Yaskawa INFORM job: A_ROOF_UPPER_0614_2_PAINT_25.JBI

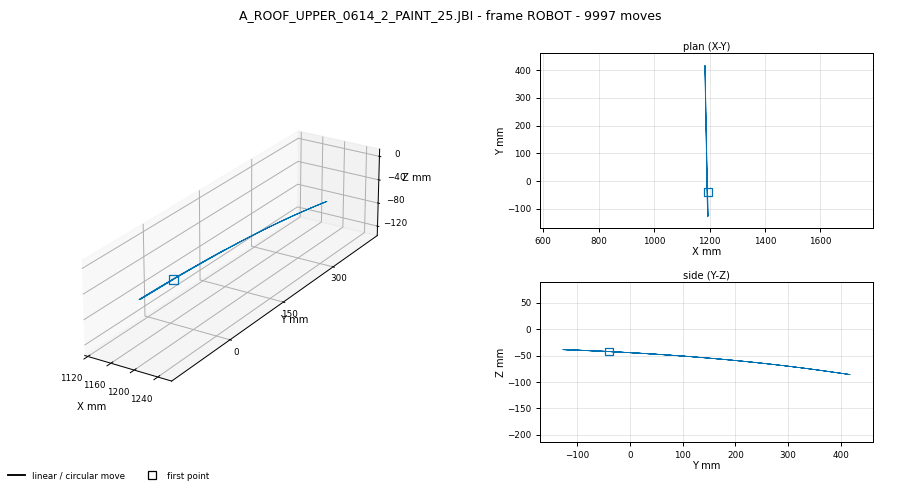
[picture p0: tool path of A_ROOF_UPPER_0614_2_PAINT_25.JBI in frame ROBOT, 9997 of 9997 moves have a stored position in this frame; points joined in program order, loops and branches not executed]
/JOB
//NAME A_ROOF_UPPER_0614_2_PAINT25
//POS
///NPOS 9997,0,0,0,0,0
///TOOL 1
///USER 0
///POSTYPE ROBOT
///RECTAN
///RCONF 1,0,0,0,0,0,0,0,0,0,0,0,0,0,0,0,0,0,0,0,0,0,0,0
C00000=1193.053,-39.607,-42.064,179.756,5.637,149.068
C00001=1193.058,-39.856,-42.051,179.753,5.636,149.068
C00002=1193.063,-40.106,-42.040,179.751,5.637,149.069
C00003=1193.068,-40.356,-42.027,179.748,5.636,149.070
C00004=1193.073,-40.606,-42.015,179.746,5.635,149.070
C00005=1193.078,-40.855,-42.002,179.744,5.636,149.071
C00006=1193.083,-41.105,-41.991,179.741,5.635,149.072
C00007=1193.088,-41.354,-41.978,179.739,5.635,149.072
C00008=1193.094,-41.604,-41.966,179.737,5.634,149.073
C00009=1193.099,-41.854,-41.954,179.735,5.634,149.074
C00010=1193.104,-42.104,-41.942,179.732,5.634,149.074
C00011=1193.110,-42.354,-41.930,179.729,5.634,149.075
C00012=1193.114,-42.603,-41.918,179.727,5.633,149.076
C00013=1193.119,-42.852,-41.906,179.725,5.633,149.076
C00014=1193.124,-43.102,-41.893,179.722,5.633,149.077
C00015=1193.130,-43.352,-41.882,179.720,5.632,149.078
C00016=1193.135,-43.602,-41.870,179.717,5.632,149.078
C00017=1193.140,-43.851,-41.857,179.715,5.632,149.079
C00018=1193.145,-44.101,-41.846,179.713,5.631,149.079
C00019=1193.151,-44.351,-41.834,179.710,5.631,149.080
C00020=1193.156,-44.600,-41.821,179.708,5.631,149.081
C00021=1193.161,-44.850,-41.809,179.705,5.631,149.082
C00022=1193.166,-45.099,-41.798,179.703,5.630,149.082
C00023=1193.171,-45.349,-41.786,179.700,5.629,149.083
C00024=1193.176,-45.599,-41.774,179.698,5.630,149.083
C00025=1193.182,-45.849,-41.762,179.696,5.629,149.084
C00026=1193.187,-46.098,-41.749,179.694,5.629,149.085
C00027=1193.192,-46.348,-41.738,179.691,5.629,149.085
C00028=1193.197,-46.597,-41.726,179.689,5.628,149.086
C00029=1193.202,-46.847,-41.713,179.686,5.628,149.087
C00030=1193.208,-47.097,-41.702,179.683,5.628,149.087
C00031=1193.212,-47.346,-41.690,179.682,5.628,149.088
C00032=1193.218,-47.596,-41.678,179.679,5.627,149.089
C00033=1193.223,-47.846,-41.666,179.677,5.627,149.089
C00034=1193.228,-48.095,-41.654,179.674,5.627,149.090
C00035=1193.233,-48.345,-41.643,179.672,5.626,149.091
C00036=1193.239,-48.594,-41.631,179.670,5.626,149.091
C00037=1193.244,-48.844,-41.619,179.667,5.625,149.092
C00038=1193.250,-49.115,-41.606,179.665,5.626,149.093
C00039=1193.255,-49.385,-41.593,179.662,5.625,149.093
C00040=1193.261,-49.655,-41.581,179.660,5.625,149.094
C00041=1193.266,-49.925,-41.568,179.657,5.624,149.095
C00042=1193.271,-50.175,-41.556,179.654,5.624,149.095
C00043=1193.276,-50.425,-41.545,179.652,5.624,149.096
C00044=1193.282,-50.674,-41.532,179.650,5.623,149.097
C00045=1193.286,-50.924,-41.521,179.647,5.623,149.097
C00046=1193.292,-51.174,-41.509,179.645,5.623,149.098
C00047=1193.298,-51.423,-41.497,179.643,5.623,149.099
C00048=1193.302,-51.672,-41.486,179.640,5.622,149.099
C00049=1193.308,-51.922,-41.474,179.638,5.622,149.100
C00050=1193.313,-52.172,-41.462,179.636,5.622,149.101
C00051=1193.318,-52.421,-41.450,179.633,5.622,149.101
C00052=1193.323,-52.671,-41.438,179.631,5.621,149.102
C00053=1193.328,-52.921,-41.426,179.629,5.621,149.102
C00054=1193.333,-53.171,-41.415,179.626,5.621,149.103
C00055=1193.339,-53.421,-41.403,179.623,5.620,149.104
C00056=1193.344,-53.670,-41.392,179.621,5.621,149.105
C00057=1193.349,-53.920,-41.380,179.619,5.620,149.105
C00058=1193.354,-54.169,-41.369,179.616,5.619,149.106
C00059=1193.359,-54.419,-41.357,179.614,5.620,149.106
C00060=1193.365,-54.669,-41.345,179.612,5.619,149.107
C00061=1193.370,-54.919,-41.334,179.609,5.618,149.108
C00062=1193.375,-55.169,-41.322,179.607,5.619,149.108
C00063=1193.380,-55.418,-41.311,179.605,5.618,149.109
C00064=1193.386,-55.667,-41.299,179.602,5.618,149.110
C00065=1193.390,-55.917,-41.288,179.600,5.617,149.110
C00066=1193.396,-56.167,-41.276,179.598,5.617,149.111
C00067=1193.401,-56.417,-41.265,179.595,5.617,149.112
C00068=1193.406,-56.667,-41.253,179.592,5.617,149.112
C00069=1193.411,-56.916,-41.242,179.590,5.617,149.113
C00070=1193.417,-57.165,-41.230,179.588,5.616,149.114
C00071=1193.422,-57.415,-41.218,179.586,5.616,149.114
C00072=1193.427,-57.665,-41.207,179.583,5.616,149.115
C00073=1193.432,-57.915,-41.195,179.581,5.616,149.116
C00074=1193.437,-58.165,-41.184,179.579,5.615,149.116
C00075=1193.443,-58.414,-41.172,179.577,5.615,149.117
C00076=1193.448,-58.663,-41.161,179.574,5.615,149.118
C00077=1193.452,-58.913,-41.150,179.571,5.614,149.118
C00078=1193.458,-59.163,-41.138,179.570,5.614,149.119
C00079=1193.462,-59.413,-41.127,179.567,5.614,149.119
C00080=1193.468,-59.662,-41.115,179.564,5.613,149.120
C00081=1193.473,-59.911,-41.104,179.562,5.614,149.121
C00082=1193.479,-60.162,-41.093,179.560,5.613,149.121
C00083=1193.484,-60.412,-41.081,179.557,5.613,149.122
C00084=1193.489,-60.662,-41.069,179.555,5.613,149.123
C00085=1193.494,-60.911,-41.058,179.553,5.612,149.123
C00086=1193.500,-61.160,-41.047,179.550,5.612,149.124
C00087=1193.504,-61.410,-41.035,179.548,5.612,149.125
C00088=1193.509,-61.660,-41.024,179.546,5.612,149.125
C00089=1193.515,-61.910,-41.013,179.543,5.611,149.126
C00090=1193.520,-62.159,-41.002,179.541,5.611,149.126
C00091=1193.526,-62.409,-40.990,179.539,5.611,149.127
C00092=1193.530,-62.659,-40.979,179.536,5.610,149.128
C00093=1193.536,-62.908,-40.967,179.534,5.611,149.129
C00094=1193.541,-63.158,-40.956,179.532,5.610,149.129
C00095=1193.546,-63.408,-40.945,179.530,5.610,149.130
C00096=1193.551,-63.658,-40.933,179.527,5.610,149.131
C00097=1193.557,-63.907,-40.923,179.524,5.609,149.131
C00098=1193.561,-64.156,-40.911,179.523,5.609,149.132
C00099=1193.567,-64.407,-40.900,179.520,5.609,149.132
C00100=1193.572,-64.656,-40.889,179.517,5.608,149.133
C00101=1193.578,-64.906,-40.877,179.515,5.609,149.134
C00102=1193.583,-65.155,-40.866,179.513,5.608,149.134
C00103=1193.588,-65.406,-40.855,179.511,5.608,149.135
C00104=1193.594,-65.655,-40.844,179.508,5.608,149.136
C00105=1193.598,-65.904,-40.833,179.506,5.607,149.136
C00106=1193.603,-66.154,-40.821,179.504,5.607,149.137
C00107=1193.609,-66.404,-40.811,179.502,5.607,149.138
C00108=1193.614,-66.654,-40.799,179.499,5.607,149.138
C00109=1193.619,-66.903,-40.788,179.496,5.606,149.139
C00110=1193.625,-67.153,-40.777,179.495,5.606,149.139
C00111=1193.630,-67.403,-40.766,179.492,5.606,149.140
C00112=1193.634,-67.652,-40.755,179.490,5.606,149.141
C00113=1193.641,-67.902,-40.744,179.487,5.606,149.142
C00114=1193.645,-68.152,-40.732,179.485,5.605,149.142
C00115=1193.650,-68.401,-40.721,179.483,5.605,149.143
C00116=1193.656,-68.651,-40.711,179.480,5.605,149.143
C00117=1193.661,-68.901,-40.699,179.478,5.604,149.144
C00118=1193.666,-69.151,-40.688,179.476,5.604,149.145
C00119=1193.671,-69.400,-40.678,179.473,5.604,149.145
C00120=1193.677,-69.650,-40.666,179.471,5.604,149.146
C00121=1193.682,-69.900,-40.655,179.469,5.604,149.147
C00122=1193.687,-70.149,-40.644,179.466,5.603,149.147
C00123=1193.692,-70.399,-40.633,179.464,5.603,149.148
C00124=1193.698,-70.649,-40.622,179.462,5.603,149.149
C00125=1193.703,-70.898,-40.611,179.459,5.603,149.149
C00126=1193.708,-71.149,-40.600,179.457,5.603,149.150
C00127=1193.713,-71.397,-40.589,179.455,5.602,149.151
C00128=1193.719,-71.648,-40.578,179.452,5.602,149.151
C00129=1193.724,-71.898,-40.567,179.450,5.602,149.152
C00130=1193.729,-72.147,-40.556,179.448,5.601,149.152
C00131=1193.734,-72.397,-40.545,179.446,5.602,149.153
C00132=1193.739,-72.646,-40.534,179.443,5.601,149.154
C00133=1193.745,-72.896,-40.523,179.441,5.600,149.154
C00134=1193.750,-73.146,-40.512,179.439,5.601,149.155
C00135=1193.755,-73.395,-40.502,179.436,5.600,149.156
C00136=1193.760,-73.645,-40.490,179.434,5.601,149.156
C00137=1193.765,-73.895,-40.480,179.432,5.600,149.157
C00138=1193.771,-74.145,-40.468,179.429,5.600,149.158
C00139=1193.776,-74.395,-40.458,179.427,5.600,149.158
C00140=1193.781,-74.644,-40.447,179.424,5.599,149.159
C00141=1193.786,-74.894,-40.436,179.422,5.599,149.160
C00142=1193.792,-75.164,-40.424,179.420,5.599,149.160
C00143=1193.798,-75.435,-40.412,179.417,5.599,149.161
C00144=1193.803,-75.707,-40.401,179.415,5.598,149.162
C00145=1193.809,-75.977,-40.389,179.412,5.598,149.162
C00146=1193.814,-76.227,-40.379,179.410,5.598,149.163
C00147=1193.820,-76.476,-40.368,179.407,5.598,149.164
C00148=1193.825,-76.726,-40.357,179.406,5.598,149.164
C00149=1193.830,-76.976,-40.345,179.403,5.597,149.165
C00150=1193.836,-77.226,-40.335,179.400,5.597,149.166
C00151=1193.841,-77.476,-40.325,179.399,5.597,149.166
C00152=1193.846,-77.725,-40.314,179.396,5.596,149.167
C00153=1193.851,-77.975,-40.303,179.394,5.597,149.168
C00154=1193.856,-78.224,-40.292,179.391,5.596,149.168
C00155=1193.861,-78.474,-40.282,179.389,5.596,149.169
C00156=1193.867,-78.724,-40.271,179.387,5.596,149.170
C00157=1193.872,-78.973,-40.260,179.384,5.596,149.170
C00158=1193.877,-79.223,-40.250,179.382,5.596,149.171
C00159=1193.882,-79.473,-40.239,179.380,5.595,149.171
C00160=1193.888,-79.722,-40.228,179.377,5.595,149.172
C00161=1193.893,-79.973,-40.217,179.375,5.595,149.173
C00162=1193.899,-80.222,-40.207,179.373,5.594,149.173
C00163=1193.904,-80.472,-40.196,179.371,5.595,149.174
C00164=1193.909,-80.721,-40.186,179.368,5.594,149.175
C00165=1193.914,-80.972,-40.175,179.366,5.594,149.175
C00166=1193.920,-81.221,-40.165,179.364,5.594,149.176
C00167=1193.924,-81.471,-40.153,179.361,5.593,149.177
C00168=1193.930,-81.720,-40.143,179.359,5.594,149.177
C00169=1193.935,-81.971,-40.133,179.357,5.593,149.178
C00170=1193.940,-82.220,-40.122,179.355,5.593,149.179
C00171=1193.945,-82.470,-40.111,179.352,5.593,149.179
C00172=1193.951,-82.719,-40.101,179.350,5.593,149.180
C00173=1193.956,-82.970,-40.090,179.348,5.593,149.180
C00174=1193.961,-83.219,-40.079,179.346,5.592,149.181
C00175=1193.966,-83.469,-40.069,179.343,5.592,149.182
C00176=1193.972,-83.718,-40.059,179.341,5.592,149.182
C00177=1193.977,-83.969,-40.048,179.339,5.591,149.183
C00178=1193.982,-84.218,-40.038,179.336,5.592,149.184
C00179=1193.988,-84.467,-40.027,179.334,5.591,149.184
C00180=1193.993,-84.717,-40.016,179.332,5.591,149.185
C00181=1193.998,-84.967,-40.006,179.330,5.591,149.186
C00182=1194.003,-85.217,-39.996,179.327,5.591,149.186
C00183=1194.009,-85.467,-39.985,179.325,5.590,149.187
C00184=1194.014,-85.716,-39.974,179.323,5.590,149.188
C00185=1194.018,-85.965,-39.964,179.321,5.590,149.188
C00186=1194.024,-86.215,-39.954,179.318,5.590,149.189
C00187=1194.029,-86.465,-39.944,179.316,5.590,149.189
C00188=1194.035,-86.715,-39.934,179.314,5.590,149.190
C00189=1194.040,-86.965,-39.923,179.311,5.589,149.191
C00190=1194.045,-87.215,-39.913,179.309,5.589,149.191
C00191=1194.050,-87.465,-39.902,179.307,5.589,149.192
C00192=1194.056,-87.714,-39.891,179.305,5.589,149.193
C00193=1194.061,-87.963,-39.881,179.302,5.588,149.193
C00194=1194.066,-88.214,-39.870,179.300,5.589,149.194
C00195=1194.072,-88.463,-39.860,179.298,5.588,149.195
C00196=1194.076,-88.713,-39.850,179.295,5.587,149.195
C00197=1194.082,-88.963,-39.840,179.293,5.588,149.196
C00198=1194.087,-89.212,-39.830,179.291,5.587,149.197
C00199=1194.092,-89.462,-39.819,179.289,5.587,149.197
C00200=1194.098,-89.712,-39.809,179.286,5.587,149.198
C00201=1194.103,-89.961,-39.799,179.284,5.587,149.199
C00202=1194.108,-90.212,-39.788,179.282,5.587,149.199
C00203=1194.113,-90.461,-39.779,179.280,5.587,149.200
C00204=1194.118,-90.711,-39.768,179.277,5.587,149.200
C00205=1194.124,-90.961,-39.758,179.275,5.586,149.201
C00206=1194.129,-91.210,-39.748,179.273,5.586,149.202
C00207=1194.134,-91.460,-39.737,179.270,5.586,149.202
C00208=1194.140,-91.710,-39.727,179.268,5.586,149.203
C00209=1194.145,-91.959,-39.717,179.266,5.585,149.204
C00210=1194.150,-92.210,-39.707,179.264,5.586,149.204
C00211=1194.155,-92.459,-39.696,179.261,5.585,149.205
C00212=1194.161,-92.709,-39.686,179.260,5.585,149.205
C00213=1194.166,-92.959,-39.676,179.257,5.585,149.206
C00214=1194.171,-93.208,-39.666,179.254,5.585,149.207
C00215=1194.177,-93.458,-39.656,179.253,5.585,149.207
C00216=1194.182,-93.708,-39.645,179.250,5.584,149.208
C00217=1194.187,-93.957,-39.635,179.248,5.584,149.209
C00218=1194.193,-94.207,-39.625,179.246,5.584,149.209
C00219=1194.197,-94.457,-39.615,179.244,5.584,149.210
C00220=1194.203,-94.706,-39.605,179.241,5.584,149.211
C00221=1194.208,-94.956,-39.594,179.240,5.584,149.211
C00222=1194.213,-95.206,-39.584,179.237,5.583,149.212
C00223=1194.218,-95.455,-39.574,179.234,5.583,149.213
C00224=1194.224,-95.705,-39.564,179.233,5.583,149.213
C00225=1194.230,-95.955,-39.555,179.230,5.582,149.214
C00226=1194.235,-96.205,-39.544,179.228,5.583,149.214
C00227=1194.239,-96.455,-39.534,179.226,5.582,149.215
C00228=1194.245,-96.704,-39.524,179.224,5.582,149.216
C00229=1194.250,-96.954,-39.514,179.221,5.582,149.216
C00230=1194.256,-97.204,-39.503,179.219,5.582,149.217
C00231=1194.260,-97.453,-39.494,179.217,5.582,149.218
C00232=1194.266,-97.703,-39.484,179.215,5.582,149.218
C00233=1194.271,-97.954,-39.474,179.212,5.581,149.219
C00234=1194.276,-98.203,-39.464,179.210,5.581,149.219
C00235=1194.282,-98.452,-39.454,179.208,5.581,149.220
C00236=1194.287,-98.702,-39.444,179.205,5.580,149.221
C00237=1194.293,-98.953,-39.434,179.203,5.581,149.221
C00238=1194.298,-99.202,-39.424,179.201,5.580,149.222
C00239=1194.303,-99.452,-39.414,179.199,5.580,149.223
C00240=1194.309,-99.701,-39.404,179.196,5.580,149.223
C00241=1194.313,-99.951,-39.394,179.194,5.580,149.224
C00242=1194.319,-100.201,-39.384,179.192,5.580,149.224
C00243=1194.325,-100.451,-39.374,179.190,5.580,149.225
C00244=1194.329,-100.700,-39.365,179.187,5.580,149.226
C00245=1194.334,-100.950,-39.354,179.186,5.580,149.226
C00246=1194.340,-101.221,-39.344,179.183,5.579,149.227
C00247=1194.346,-101.493,-39.333,179.180,5.579,149.228
C00248=1194.352,-101.765,-39.322,179.178,5.579,149.229
C00249=1194.357,-102.036,-39.311,179.176,5.579,149.229
C00250=1194.363,-102.286,-39.301,179.173,5.578,149.230
C00251=1194.368,-102.536,-39.292,179.171,5.578,149.230
C00252=1194.373,-102.785,-39.282,179.169,5.578,149.231
C00253=1194.379,-103.035,-39.272,179.167,5.578,149.232
C00254=1194.384,-103.285,-39.263,179.164,5.578,149.232
C00255=1194.389,-103.535,-39.252,179.162,5.578,149.233
C00256=1194.394,-103.784,-39.243,179.160,5.577,149.234
C00257=1194.400,-104.034,-39.233,179.158,5.578,149.234
C00258=1194.406,-104.284,-39.223,179.155,5.577,149.235
C00259=1194.410,-104.534,-39.213,179.154,5.577,149.235
C00260=1194.416,-104.784,-39.204,179.151,5.577,149.236
C00261=1194.421,-105.033,-39.194,179.149,5.577,149.237
C00262=1194.426,-105.283,-39.184,179.147,5.576,149.237
C00263=1194.431,-105.532,-39.175,179.145,5.577,149.238
C00264=1194.437,-105.782,-39.165,179.143,5.576,149.239
C00265=1194.441,-106.032,-39.155,179.140,5.576,149.239
C00266=1194.447,-106.282,-39.145,179.138,5.576,149.240
C00267=1194.452,-106.531,-39.136,179.136,5.576,149.240
C00268=1194.458,-106.782,-39.126,179.133,5.576,149.241
C00269=1194.463,-107.031,-39.116,179.131,5.575,149.242
C00270=1194.468,-107.280,-39.106,179.129,5.575,149.242
C00271=1194.474,-107.531,-39.096,179.127,5.575,149.243
C00272=1194.479,-107.780,-39.087,179.125,5.575,149.244
C00273=1194.484,-108.031,-39.077,179.122,5.574,149.244
C00274=1194.489,-108.280,-39.068,179.120,5.575,149.245
C00275=1194.495,-108.530,-39.058,179.118,5.574,149.246
C00276=1194.500,-108.779,-39.049,179.116,5.574,149.246
C00277=1194.506,-109.029,-39.039,179.114,5.574,149.247
C00278=1194.511,-109.279,-39.029,179.112,5.574,149.247
C00279=1194.516,-109.529,-39.019,179.109,5.574,149.248
C00280=1194.521,-109.779,-39.010,179.107,5.574,149.249
C00281=1194.526,-110.028,-39.000,179.105,5.573,149.249
C00282=1194.532,-110.278,-38.991,179.103,5.574,149.250
C00283=1194.537,-110.527,-38.981,179.100,5.573,149.251
C00284=1194.542,-110.777,-38.972,179.098,5.573,149.251
C00285=1194.547,-111.027,-38.962,179.096,5.572,149.252
C00286=1194.553,-111.277,-38.953,179.094,5.573,149.252
C00287=1194.558,-111.527,-38.944,179.091,5.572,149.253
C00288=1194.564,-111.776,-38.934,179.090,5.572,149.254
C00289=1194.569,-112.027,-38.924,179.087,5.572,149.254
C00290=1194.574,-112.276,-38.914,179.085,5.572,149.255
C00291=1194.579,-112.526,-38.905,179.083,5.572,149.256
C00292=1194.584,-112.775,-38.896,179.081,5.572,149.256
C00293=1194.590,-113.026,-38.886,179.078,5.571,149.257
C00294=1194.595,-113.275,-38.876,179.076,5.572,149.257
C00295=1194.601,-113.525,-38.867,179.074,5.571,149.258
C00296=1194.606,-113.775,-38.858,179.072,5.571,149.259
C00297=1194.611,-114.024,-38.848,179.069,5.571,149.259
C00298=1194.617,-114.274,-38.839,179.068,5.571,149.260
C00299=1194.622,-114.523,-38.829,179.065,5.571,149.261
C00300=1194.628,-114.774,-38.820,179.064,5.571,149.261
C00301=1194.633,-115.023,-38.811,179.061,5.570,149.262
C00302=1194.638,-115.273,-38.801,179.059,5.571,149.263
C00303=1194.644,-115.523,-38.792,179.057,5.570,149.263
C00304=1194.649,-115.773,-38.783,179.055,5.570,149.264
C00305=1194.654,-116.022,-38.773,179.052,5.569,149.264
C00306=1194.659,-116.272,-38.764,179.050,5.570,149.265
C00307=1194.665,-116.522,-38.755,179.048,5.569,149.266
C00308=1194.670,-116.772,-38.745,179.046,5.569,149.266
C00309=1194.675,-117.021,-38.736,179.043,5.569,149.267
C00310=1194.680,-117.272,-38.727,179.042,5.569,149.267
C00311=1194.686,-117.521,-38.716,179.039,5.569,149.268
C00312=1194.691,-117.771,-38.707,179.037,5.569,149.269
C00313=1194.696,-118.021,-38.699,179.035,5.568,149.269
C00314=1194.701,-118.270,-38.689,179.033,5.569,149.270
C00315=1194.707,-118.521,-38.679,179.030,5.568,149.270
C00316=1194.712,-118.770,-38.671,179.028,5.568,149.271
C00317=1194.717,-119.020,-38.662,179.027,5.568,149.272
C00318=1194.723,-119.270,-38.651,179.024,5.568,149.272
C00319=1194.728,-119.520,-38.643,179.022,5.568,149.273
C00320=1194.733,-119.770,-38.634,179.020,5.568,149.274
C00321=1194.738,-120.019,-38.624,179.018,5.568,149.274
C00322=1194.744,-120.269,-38.615,179.016,5.567,149.275
C00323=1194.749,-120.518,-38.606,179.013,5.568,149.275
C00324=1194.755,-120.768,-38.597,179.011,5.567,149.276
C00325=1194.761,-121.018,-38.588,179.009,5.567,149.277
C00326=1194.765,-121.267,-38.578,179.006,5.567,149.277
C00327=1194.771,-121.517,-38.569,179.005,5.567,149.278
C00328=1194.776,-121.767,-38.560,179.002,5.566,149.279
C00329=1194.782,-122.017,-38.551,179.001,5.566,149.279
C00330=1194.787,-122.267,-38.542,178.998,5.566,149.280
C00331=1194.792,-122.516,-38.532,178.996,5.566,149.280
C00332=1194.797,-122.766,-38.523,178.994,5.566,149.281
C00333=1194.802,-123.016,-38.514,178.992,5.566,149.282
C00334=1194.808,-123.266,-38.505,178.989,5.565,149.282
C00335=1194.813,-123.516,-38.496,178.987,5.566,149.283
C00336=1194.818,-123.766,-38.487,178.985,5.565,149.283
C00337=1194.823,-124.015,-38.478,178.983,5.565,149.284
C00338=1194.829,-124.265,-38.468,178.981,5.565,149.285
C00339=1194.834,-124.515,-38.459,178.979,5.565,149.285
C00340=1194.839,-124.765,-38.450,178.977,5.565,149.286
C00341=1194.844,-125.015,-38.441,178.974,5.565,149.287
C00342=1194.850,-125.264,-38.433,178.972,5.565,149.287
C00343=1194.855,-125.514,-38.424,178.970,5.564,149.288
C00344=1194.861,-125.764,-38.414,178.968,5.565,149.288
C00345=1194.866,-126.013,-38.405,178.966,5.564,149.289
C00346=1194.871,-126.263,-38.396,178.964,5.564,149.290
C00347=1194.876,-126.513,-38.387,178.962,5.563,149.290
C00348=1194.882,-126.763,-38.378,178.960,5.564,149.291
C00349=1194.887,-127.013,-38.369,178.957,5.563,149.291
C00350=1194.466,-127.024,-38.408,178.953,5.567,149.293
C00351=1194.460,-126.774,-38.417,178.956,5.567,149.293
C00352=1194.455,-126.524,-38.426,178.958,5.567,149.292
C00353=1194.450,-126.274,-38.435,178.960,5.567,149.292
C00354=1194.445,-126.024,-38.444,178.962,5.567,149.291
C00355=1194.440,-125.775,-38.453,178.964,5.568,149.290
C00356=1194.434,-125.525,-38.463,178.966,5.567,149.290
C00357=1194.429,-125.275,-38.472,178.968,5.568,149.289
C00358=1194.423,-125.026,-38.480,178.971,5.568,149.288
C00359=1194.418,-124.776,-38.489,178.973,5.569,149.288
C00360=1194.413,-124.526,-38.498,178.975,5.568,149.287
C00361=1194.407,-124.276,-38.507,178.977,5.569,149.287
C00362=1194.402,-124.026,-38.516,178.979,5.568,149.286
C00363=1194.397,-123.776,-38.525,178.982,5.569,149.285
C00364=1194.392,-123.527,-38.535,178.983,5.569,149.285
C00365=1194.387,-123.277,-38.544,178.985,5.568,149.284
C00366=1194.381,-123.027,-38.553,178.988,5.569,149.284
C00367=1194.376,-122.777,-38.562,178.990,5.569,149.283
C00368=1194.370,-122.527,-38.571,178.992,5.570,149.282
C00369=1194.365,-122.277,-38.580,178.994,5.569,149.282
C00370=1194.360,-122.028,-38.590,178.996,5.570,149.281
C00371=1194.354,-121.778,-38.599,178.998,5.570,149.280
C00372=1194.349,-121.528,-38.608,179.001,5.570,149.280
C00373=1194.344,-121.278,-38.617,179.003,5.570,149.279
C00374=1194.338,-121.028,-38.626,179.005,5.570,149.279
C00375=1194.333,-120.779,-38.636,179.007,5.570,149.278
C00376=1194.328,-120.530,-38.644,179.010,5.571,149.277
C00377=1194.322,-120.280,-38.653,179.011,5.571,149.277
C00378=1194.316,-120.030,-38.663,179.014,5.571,149.276
C00379=1194.312,-119.780,-38.672,179.016,5.571,149.275
C00380=1194.306,-119.531,-38.681,179.018,5.571,149.275
C00381=1194.301,-119.281,-38.690,179.020,5.571,149.274
C00382=1194.295,-119.031,-38.700,179.022,5.572,149.274
C00383=1194.291,-118.781,-38.709,179.024,5.571,149.273
C00384=1194.285,-118.532,-38.718,179.027,5.572,149.273
C00385=1194.279,-118.281,-38.728,179.029,5.572,149.272
C00386=1194.274,-118.032,-38.737,179.031,5.572,149.271
C00387=1194.269,-117.782,-38.746,179.033,5.572,149.271
C00388=1194.264,-117.532,-38.755,179.036,5.573,149.270
C00389=1194.258,-117.282,-38.765,179.037,5.573,149.269
C00390=1194.253,-117.033,-38.774,179.040,5.573,149.269
C00391=1194.248,-116.783,-38.783,179.042,5.573,149.268
C00392=1194.242,-116.533,-38.793,179.044,5.573,149.267
C00393=1194.238,-116.284,-38.802,179.046,5.573,149.267
C00394=1194.232,-116.033,-38.812,179.048,5.573,149.266
C00395=1194.227,-115.783,-38.821,179.051,5.573,149.266
C00396=1194.222,-115.534,-38.831,179.052,5.573,149.265
C00397=1194.216,-115.284,-38.840,179.055,5.574,149.264
C00398=1194.211,-115.034,-38.849,179.057,5.573,149.264
C00399=1194.206,-114.785,-38.859,179.059,5.574,149.263
C00400=1194.200,-114.534,-38.868,179.061,5.574,149.262
C00401=1194.196,-114.285,-38.878,179.063,5.575,149.262
C00402=1194.190,-114.035,-38.887,179.066,5.574,149.261
C00403=1194.184,-113.785,-38.896,179.068,5.574,149.261
C00404=1194.180,-113.536,-38.906,179.070,5.574,149.260
C00405=1194.174,-113.286,-38.915,179.072,5.575,149.259
C00406=1194.169,-113.037,-38.925,179.074,5.575,149.259
C00407=1194.163,-112.786,-38.934,179.077,5.575,149.258
C00408=1194.158,-112.537,-38.943,179.079,5.575,149.257
C00409=1194.153,-112.287,-38.953,179.081,5.576,149.257
C00410=1194.147,-112.037,-38.962,179.083,5.575,149.256
C00411=1194.142,-111.788,-38.972,179.085,5.576,149.256
C00412=1194.136,-111.538,-38.981,179.087,5.576,149.255
C00413=1194.132,-111.288,-38.991,179.090,5.576,149.254
C00414=1194.126,-111.038,-39.001,179.092,5.576,149.254
C00415=1194.121,-110.788,-39.011,179.094,5.576,149.253
C00416=1194.116,-110.539,-39.019,179.096,5.576,149.253
C00417=1194.110,-110.289,-39.030,179.099,5.577,149.252
C00418=1194.105,-110.039,-39.039,179.101,5.576,149.251
C00419=1194.100,-109.790,-39.049,179.103,5.577,149.251
C00420=1194.095,-109.540,-39.058,179.106,5.578,149.250
C00421=1194.089,-109.290,-39.068,179.107,5.578,149.250
C00422=1194.084,-109.040,-39.077,179.110,5.578,149.249
C00423=1194.079,-108.790,-39.087,179.112,5.578,149.248
C00424=1194.074,-108.540,-39.096,179.114,5.578,149.248
C00425=1194.068,-108.291,-39.106,179.116,5.578,149.247
C00426=1194.063,-108.041,-39.115,179.118,5.579,149.246
C00427=1194.057,-107.791,-39.126,179.120,5.578,149.246
C00428=1194.052,-107.542,-39.134,179.123,5.579,149.245
C00429=1194.046,-107.292,-39.145,179.125,5.579,149.244
C00430=1194.042,-107.042,-39.155,179.127,5.579,149.244
C00431=1194.036,-106.792,-39.164,179.130,5.579,149.243
C00432=1194.031,-106.543,-39.174,179.132,5.580,149.243
C00433=1194.026,-106.292,-39.183,179.134,5.579,149.242
C00434=1194.021,-106.043,-39.193,179.136,5.580,149.241
C00435=1194.015,-105.794,-39.203,179.138,5.580,149.241
C00436=1194.010,-105.544,-39.212,179.141,5.580,149.240
C00437=1194.005,-105.294,-39.223,179.142,5.580,149.239
C00438=1193.999,-105.043,-39.232,179.145,5.580,149.239
C00439=1193.994,-104.794,-39.242,179.147,5.580,149.238
C00440=1193.989,-104.545,-39.252,179.149,5.581,149.238
C00441=1193.983,-104.295,-39.261,179.151,5.580,149.237
C00442=1193.978,-104.045,-39.271,179.154,5.581,149.236
C00443=1193.974,-103.795,-39.281,179.156,5.581,149.236
C00444=1193.968,-103.545,-39.290,179.158,5.581,149.235
C00445=1193.962,-103.296,-39.301,179.160,5.581,149.234
C00446=1193.957,-103.046,-39.310,179.163,5.582,149.234
C00447=1193.952,-102.796,-39.320,179.165,5.581,149.233
C00448=1193.947,-102.546,-39.330,179.167,5.582,149.233
C00449=1193.941,-102.297,-39.340,179.170,5.582,149.232
C00450=1193.935,-102.047,-39.349,179.172,5.582,149.231
C00451=1193.930,-101.775,-39.360,179.174,5.582,149.230
C00452=1193.925,-101.504,-39.371,179.176,5.582,149.230
C00453=1193.918,-101.232,-39.382,179.179,5.583,149.229
C00454=1193.913,-100.961,-39.393,179.181,5.583,149.228
C00455=1193.907,-100.711,-39.402,179.183,5.583,149.228
C00456=1193.903,-100.461,-39.412,179.186,5.584,149.227
C00457=1193.897,-100.212,-39.422,179.188,5.583,149.227
C00458=1193.892,-99.962,-39.433,179.190,5.584,149.226
C00459=1193.887,-99.713,-39.442,179.192,5.584,149.225
C00460=1193.882,-99.462,-39.452,179.195,5.584,149.225
C00461=1193.877,-99.213,-39.462,179.197,5.584,149.224
C00462=1193.871,-98.963,-39.472,179.199,5.584,149.223
C00463=1193.866,-98.714,-39.482,179.202,5.585,149.223
C00464=1193.860,-98.463,-39.492,179.204,5.584,149.222
C00465=1193.855,-98.213,-39.502,179.206,5.585,149.222
C00466=1193.850,-97.964,-39.512,179.208,5.585,149.221
C00467=1193.844,-97.714,-39.522,179.211,5.585,149.220
C00468=1193.840,-97.464,-39.532,179.212,5.585,149.220
C00469=1193.834,-97.215,-39.542,179.215,5.586,149.219
C00470=1193.828,-96.965,-39.552,179.217,5.585,149.218
C00471=1193.823,-96.715,-39.562,179.219,5.586,149.218
C00472=1193.819,-96.465,-39.572,179.221,5.586,149.217
C00473=1193.813,-96.216,-39.582,179.224,5.586,149.216
C00474=1193.807,-95.966,-39.592,179.226,5.587,149.216
C00475=1193.803,-95.716,-39.602,179.228,5.586,149.215
C00476=1193.797,-95.467,-39.612,179.231,5.587,149.214
C00477=1193.792,-95.217,-39.623,179.232,5.587,149.214
C00478=1193.786,-94.967,-39.632,179.235,5.587,149.213
C00479=1193.782,-94.717,-39.642,179.237,5.587,149.213
C00480=1193.776,-94.468,-39.652,179.239,5.588,149.212
C00481=1193.771,-94.218,-39.663,179.241,5.587,149.211
C00482=1193.766,-93.968,-39.673,179.244,5.588,149.211
C00483=1193.760,-93.718,-39.683,179.246,5.588,149.210
C00484=1193.755,-93.469,-39.693,179.248,5.588,149.209
C00485=1193.750,-93.219,-39.704,179.251,5.588,149.209
C00486=1193.744,-92.969,-39.714,179.253,5.588,149.208
C00487=1193.739,-92.720,-39.724,179.255,5.589,149.207
C00488=1193.734,-92.469,-39.735,179.257,5.588,149.207
C00489=1193.729,-92.220,-39.744,179.260,5.589,149.206
C00490=1193.723,-91.971,-39.754,179.262,5.589,149.206
C00491=1193.718,-91.720,-39.765,179.264,5.589,149.205
C00492=1193.713,-91.471,-39.775,179.266,5.589,149.204
C00493=1193.707,-91.221,-39.785,179.269,5.590,149.204
C00494=1193.703,-90.971,-39.795,179.271,5.590,149.203
C00495=1193.697,-90.722,-39.806,179.273,5.590,149.202
C00496=1193.692,-90.472,-39.816,179.276,5.591,149.202
C00497=1193.687,-90.222,-39.826,179.278,5.590,149.201
C00498=1193.681,-89.972,-39.837,179.280,5.591,149.201
C00499=1193.676,-89.723,-39.847,179.282,5.591,149.200
C00500=1193.671,-89.473,-39.857,179.285,5.591,149.199
C00501=1193.666,-89.223,-39.867,179.287,5.591,149.198
C00502=1193.661,-88.973,-39.877,179.289,5.591,149.198
C00503=1193.655,-88.724,-39.888,179.292,5.592,149.197
C00504=1193.650,-88.474,-39.898,179.294,5.591,149.197
C00505=1193.645,-88.224,-39.908,179.296,5.592,149.196
C00506=1193.639,-87.974,-39.919,179.298,5.592,149.195
C00507=1193.634,-87.724,-39.929,179.301,5.592,149.195
C00508=1193.629,-87.475,-39.940,179.303,5.593,149.194
C00509=1193.624,-87.226,-39.950,179.305,5.593,149.193
C00510=1193.619,-86.976,-39.960,179.308,5.593,149.193
C00511=1193.613,-86.726,-39.971,179.309,5.593,149.192
C00512=1193.608,-86.476,-39.981,179.312,5.593,149.192
C00513=1193.603,-86.226,-39.991,179.314,5.593,149.191
C00514=1193.597,-85.977,-40.002,179.317,5.594,149.190
C00515=1193.592,-85.727,-40.012,179.319,5.594,149.190
C00516=1193.587,-85.478,-40.023,179.321,5.594,149.189
C00517=1193.582,-85.227,-40.034,179.324,5.594,149.188
C00518=1193.576,-84.978,-40.044,179.325,5.594,149.188
C00519=1193.571,-84.728,-40.054,179.328,5.595,149.187
C00520=1193.565,-84.478,-40.065,179.330,5.594,149.186
C00521=1193.561,-84.228,-40.076,179.332,5.595,149.186
C00522=1193.555,-83.979,-40.086,179.335,5.596,149.185
C00523=1193.550,-83.729,-40.096,179.337,5.595,149.184
C00524=1193.545,-83.479,-40.107,179.339,5.596,149.184
C00525=1193.539,-83.230,-40.117,179.341,5.596,149.183
C00526=1193.534,-82.980,-40.128,179.344,5.596,149.183
C00527=1193.529,-82.730,-40.139,179.346,5.596,149.182
C00528=1193.524,-82.480,-40.149,179.348,5.596,149.181
C00529=1193.518,-82.231,-40.159,179.351,5.597,149.181
C00530=1193.513,-81.981,-40.171,179.353,5.597,149.180
C00531=1193.508,-81.731,-40.181,179.355,5.597,149.179
C00532=1193.503,-81.481,-40.191,179.357,5.597,149.179
C00533=1193.497,-81.232,-40.202,179.360,5.597,149.178
C00534=1193.493,-80.982,-40.213,179.362,5.598,149.177
C00535=1193.487,-80.732,-40.223,179.364,5.598,149.177
C00536=1193.482,-80.482,-40.234,179.367,5.598,149.176
C00537=1193.477,-80.233,-40.245,179.369,5.598,149.175
C00538=1193.472,-79.983,-40.255,179.371,5.599,149.175
C00539=1193.466,-79.734,-40.265,179.374,5.599,149.174
C00540=1193.461,-79.484,-40.277,179.376,5.599,149.174
C00541=1193.456,-79.234,-40.287,179.378,5.599,149.173
C00542=1193.451,-78.984,-40.298,179.380,5.599,149.172
C00543=1193.445,-78.735,-40.308,179.383,5.600,149.172
C00544=1193.440,-78.485,-40.319,179.385,5.600,149.171
C00545=1193.435,-78.235,-40.329,179.387,5.600,149.170
C00546=1193.430,-77.986,-40.341,179.390,5.600,149.170
C00547=1193.425,-77.736,-40.351,179.392,5.600,149.169
C00548=1193.419,-77.486,-40.362,179.394,5.600,149.168
C00549=1193.414,-77.237,-40.373,179.397,5.601,149.168
C00550=1193.409,-76.987,-40.383,179.399,5.601,149.167
C00551=1193.403,-76.738,-40.394,179.401,5.601,149.166
C00552=1193.398,-76.487,-40.405,179.403,5.601,149.166
C00553=1193.393,-76.237,-40.415,179.406,5.602,149.165
C00554=1193.388,-75.988,-40.426,179.408,5.602,149.165
C00555=1193.382,-75.717,-40.439,179.410,5.602,149.164
C00556=1193.376,-75.446,-40.450,179.413,5.602,149.163
C00557=1193.371,-75.176,-40.461,179.416,5.603,149.162
C00558=1193.365,-74.905,-40.474,179.418,5.603,149.162
C00559=1193.360,-74.655,-40.484,179.420,5.603,149.161
C00560=1193.355,-74.405,-40.495,179.423,5.603,149.160
C00561=1193.349,-74.156,-40.506,179.425,5.604,149.160
C00562=1193.344,-73.906,-40.517,179.427,5.603,149.159
C00563=1193.339,-73.656,-40.528,179.430,5.604,149.159
C00564=1193.334,-73.407,-40.539,179.432,5.604,149.158
C00565=1193.329,-73.157,-40.549,179.434,5.604,149.157
C00566=1193.323,-72.907,-40.561,179.437,5.605,149.156
C00567=1193.318,-72.657,-40.572,179.439,5.605,149.156
C00568=1193.312,-72.408,-40.582,179.441,5.605,149.155
C00569=1193.307,-72.158,-40.593,179.443,5.605,149.155
C00570=1193.303,-71.908,-40.604,179.445,5.606,149.154
C00571=1193.296,-71.658,-40.615,179.448,5.606,149.153
C00572=1193.292,-71.409,-40.626,179.450,5.606,149.153
C00573=1193.287,-71.159,-40.637,179.453,5.606,149.152
C00574=1193.281,-70.910,-40.648,179.455,5.607,149.151
C00575=1193.276,-70.659,-40.659,179.457,5.607,149.151
C00576=1193.270,-70.410,-40.670,179.460,5.607,149.150
C00577=1193.266,-70.161,-40.681,179.462,5.607,149.149
C00578=1193.261,-69.910,-40.692,179.464,5.607,149.149
C00579=1193.255,-69.661,-40.703,179.467,5.608,149.148
C00580=1193.250,-69.411,-40.714,179.469,5.607,149.147
C00581=1193.245,-69.161,-40.725,179.472,5.608,149.147
C00582=1193.240,-68.912,-40.736,179.474,5.609,149.146
C00583=1193.234,-68.662,-40.747,179.476,5.608,149.146
C00584=1193.229,-68.412,-40.759,179.478,5.609,149.145
C00585=1193.224,-68.163,-40.770,179.481,5.610,149.144
C00586=1193.218,-67.913,-40.781,179.483,5.609,149.144
C00587=1193.214,-67.663,-40.792,179.485,5.610,149.143
C00588=1193.208,-67.414,-40.803,179.487,5.609,149.142
C00589=1193.203,-67.164,-40.814,179.490,5.610,149.142
C00590=1193.198,-66.914,-40.825,179.492,5.610,149.141
C00591=1193.193,-66.665,-40.836,179.494,5.610,149.140
C00592=1193.187,-66.414,-40.847,179.497,5.611,149.140
C00593=1193.182,-66.165,-40.859,179.499,5.611,149.139
C00594=1193.177,-65.916,-40.870,179.501,5.611,149.138
C00595=1193.171,-65.665,-40.881,179.504,5.611,149.138
C00596=1193.166,-65.416,-40.892,179.507,5.612,149.137
C00597=1193.161,-65.167,-40.903,179.508,5.612,149.137
C00598=1193.156,-64.917,-40.915,179.511,5.612,149.136
C00599=1193.151,-64.667,-40.926,179.514,5.613,149.135
C00600=1193.146,-64.417,-40.937,179.516,5.612,149.134
C00601=1193.140,-64.168,-40.948,179.518,5.613,149.134
C00602=1193.135,-63.918,-40.960,179.520,5.613,149.133
C00603=1193.130,-63.668,-40.970,179.523,5.613,149.133
C00604=1193.124,-63.419,-40.982,179.525,5.614,149.132
C00605=1193.120,-63.169,-40.993,179.527,5.614,149.131
C00606=1193.114,-62.919,-41.005,179.530,5.614,149.131
C00607=1193.109,-62.669,-41.016,179.532,5.615,149.130
C00608=1193.104,-62.420,-41.026,179.534,5.614,149.129
C00609=1193.098,-62.170,-41.038,179.537,5.615,149.129
C00610=1193.094,-61.920,-41.050,179.539,5.615,149.128
C00611=1193.088,-61.670,-41.061,179.541,5.615,149.127
C00612=1193.083,-61.421,-41.072,179.544,5.615,149.127
C00613=1193.077,-61.171,-41.084,179.546,5.616,149.126
C00614=1193.073,-60.921,-41.095,179.548,5.616,149.126
C00615=1193.068,-60.672,-41.106,179.551,5.616,149.125
C00616=1193.062,-60.422,-41.118,179.554,5.617,149.124
C00617=1193.057,-60.173,-41.129,179.555,5.617,149.124
C00618=1193.052,-59.923,-41.141,179.558,5.617,149.123
C00619=1193.047,-59.673,-41.152,179.560,5.618,149.122
C00620=1193.042,-59.423,-41.164,179.563,5.617,149.122
C00621=1193.036,-59.174,-41.175,179.565,5.618,149.121
C00622=1193.031,-58.924,-41.186,179.567,5.619,149.120
C00623=1193.026,-58.674,-41.197,179.569,5.618,149.120
C00624=1193.020,-58.424,-41.209,179.572,5.619,149.119
C00625=1193.016,-58.175,-41.221,179.574,5.619,149.118
C00626=1193.010,-57.925,-41.232,179.576,5.619,149.118
C00627=1193.005,-57.676,-41.243,179.579,5.620,149.117
C00628=1193.000,-57.426,-41.255,179.582,5.620,149.116
C00629=1192.995,-57.176,-41.267,179.584,5.620,149.116
C00630=1192.989,-56.926,-41.278,179.586,5.620,149.115
C00631=1192.985,-56.677,-41.290,179.589,5.621,149.114
C00632=1192.979,-56.427,-41.301,179.591,5.620,149.114
C00633=1192.974,-56.178,-41.313,179.593,5.621,149.113
C00634=1192.969,-55.928,-41.324,179.596,5.622,149.113
C00635=1192.964,-55.678,-41.336,179.598,5.621,149.112
C00636=1192.959,-55.428,-41.348,179.600,5.622,149.111
C00637=1192.954,-55.179,-41.359,179.603,5.622,149.110
C00638=1192.948,-54.929,-41.370,179.605,5.623,149.110
C00639=1192.943,-54.680,-41.382,179.607,5.623,149.109
C00640=1192.938,-54.430,-41.394,179.610,5.623,149.109
C00641=1192.932,-54.180,-41.405,179.613,5.624,149.108
C00642=1192.928,-53.930,-41.417,179.614,5.624,149.107
C00643=1192.922,-53.680,-41.429,179.617,5.624,149.107
C00644=1192.917,-53.431,-41.440,179.620,5.624,149.106
C00645=1192.912,-53.181,-41.452,179.622,5.624,149.105
C00646=1192.907,-52.932,-41.463,179.624,5.625,149.105
C00647=1192.902,-52.683,-41.475,179.626,5.625,149.104
C00648=1192.896,-52.433,-41.487,179.629,5.625,149.103
C00649=1192.891,-52.183,-41.499,179.631,5.625,149.103
C00650=1192.886,-51.933,-41.510,179.634,5.626,149.102
C00651=1192.881,-51.683,-41.522,179.636,5.627,149.102
C00652=1192.876,-51.433,-41.534,179.638,5.626,149.101
C00653=1192.870,-51.184,-41.545,179.641,5.627,149.100
C00654=1192.866,-50.934,-41.557,179.643,5.627,149.099
C00655=1192.860,-50.685,-41.569,179.645,5.627,149.099
C00656=1192.855,-50.435,-41.581,179.648,5.628,149.098
C00657=1192.850,-50.186,-41.592,179.650,5.628,149.098
C00658=1192.845,-49.936,-41.604,179.652,5.628,149.097
C00659=1192.839,-49.665,-41.617,179.655,5.628,149.096
C00660=1192.833,-49.396,-41.630,179.658,5.629,149.095
C00661=1192.828,-49.125,-41.643,179.660,5.629,149.095
C00662=1192.823,-48.855,-41.656,179.663,5.630,149.094
C00663=1192.817,-48.605,-41.667,179.665,5.630,149.094
C00664=1192.812,-48.355,-41.679,179.667,5.630,149.093
C00665=1192.807,-48.106,-41.690,179.670,5.630,149.092
C00666=1192.801,-47.856,-41.702,179.673,5.631,149.091
C00667=1192.796,-47.607,-41.715,179.675,5.631,149.091
C00668=1192.791,-47.357,-41.727,179.677,5.631,149.090
C00669=1192.786,-47.107,-41.738,179.680,5.632,149.090
C00670=1192.780,-46.858,-41.750,179.682,5.631,149.089
C00671=1192.775,-46.608,-41.762,179.684,5.632,149.088
C00672=1192.770,-46.358,-41.774,179.687,5.633,149.088
C00673=1192.765,-46.109,-41.786,179.689,5.633,149.087
C00674=1192.760,-45.859,-41.798,179.691,5.633,149.086
C00675=1192.755,-45.609,-41.810,179.694,5.633,149.086
C00676=1192.749,-45.359,-41.822,179.697,5.634,149.085
C00677=1192.745,-45.110,-41.834,179.699,5.635,149.084
C00678=1192.739,-44.861,-41.846,179.701,5.634,149.084
C00679=1192.734,-44.611,-41.858,179.704,5.635,149.083
C00680=1192.729,-44.361,-41.870,179.706,5.635,149.082
C00681=1192.723,-44.111,-41.882,179.708,5.635,149.082
C00682=1192.719,-43.862,-41.893,179.710,5.636,149.081
C00683=1192.714,-43.612,-41.906,179.713,5.636,149.080
C00684=1192.708,-43.362,-41.918,179.716,5.636,149.080
C00685=1192.703,-43.113,-41.930,179.717,5.636,149.079
C00686=1192.698,-42.863,-41.942,179.720,5.637,149.079
C00687=1192.693,-42.614,-41.954,179.723,5.637,149.078
C00688=1192.688,-42.364,-41.966,179.725,5.638,149.077
C00689=1192.682,-42.114,-41.978,179.727,5.637,149.076
C00690=1192.677,-41.864,-41.990,179.730,5.638,149.076
C00691=1192.672,-41.615,-42.003,179.732,5.639,149.075
C00692=1192.666,-41.365,-42.015,179.734,5.638,149.075
C00693=1192.662,-41.116,-42.027,179.737,5.639,149.074
C00694=1192.657,-40.866,-42.038,179.739,5.640,149.073
C00695=1192.651,-40.617,-42.051,179.742,5.640,149.073
C00696=1192.646,-40.367,-42.063,179.744,5.640,149.072
C00697=1192.641,-40.116,-42.075,179.747,5.640,149.071
C00698=1192.636,-39.867,-42.088,179.749,5.641,149.071
C00699=1192.631,-39.617,-42.100,179.752,5.641,149.070
C00700=1192.625,-39.368,-42.112,179.754,5.641,149.069
C00701=1192.621,-39.118,-42.124,179.756,5.642,149.069
C00702=1192.616,-38.869,-42.136,179.759,5.642,149.068
C00703=1192.610,-38.619,-42.148,179.761,5.643,149.068
C00704=1192.605,-38.370,-42.161,179.763,5.643,149.067
C00705=1192.600,-38.120,-42.173,179.766,5.643,149.066
C00706=1192.595,-37.870,-42.185,179.768,5.643,149.065
C00707=1192.589,-37.620,-42.197,179.771,5.644,149.065
C00708=1192.584,-37.371,-42.210,179.773,5.644,149.064
C00709=1192.579,-37.122,-42.222,179.775,5.644,149.064
C00710=1192.574,-36.871,-42.235,179.778,5.645,149.063
C00711=1192.569,-36.622,-42.247,179.781,5.645,149.062
C00712=1192.563,-36.372,-42.259,179.783,5.645,149.061
C00713=1192.558,-36.122,-42.272,179.785,5.646,149.061
C00714=1192.553,-35.873,-42.283,179.788,5.646,149.060
C00715=1192.548,-35.623,-42.296,179.790,5.647,149.060
C00716=1192.543,-35.374,-42.309,179.792,5.646,149.059
C00717=1192.537,-35.124,-42.321,179.795,5.647,149.058
C00718=1192.532,-34.875,-42.333,179.797,5.648,149.058
C00719=1192.528,-34.625,-42.346,179.800,5.648,149.057
C00720=1192.522,-34.375,-42.358,179.803,5.648,149.056
C00721=1192.517,-34.125,-42.371,179.805,5.648,149.056
C00722=1192.512,-33.875,-42.383,179.807,5.649,149.055
C00723=1192.507,-33.626,-42.395,179.809,5.649,149.054
C00724=1192.501,-33.377,-42.408,179.812,5.650,149.054
C00725=1192.496,-33.127,-42.420,179.814,5.650,149.053
C00726=1192.491,-32.877,-42.433,179.816,5.650,149.053
C00727=1192.486,-32.628,-42.445,179.819,5.651,149.052
C00728=1192.481,-32.378,-42.458,179.822,5.651,149.051
C00729=1192.476,-32.128,-42.470,179.824,5.651,149.050
C00730=1192.471,-31.879,-42.482,179.826,5.651,149.050
C00731=1192.466,-31.630,-42.495,179.829,5.652,149.049
C00732=1192.461,-31.379,-42.507,179.831,5.653,149.049
C00733=1192.456,-31.130,-42.520,179.834,5.653,149.048
C00734=1192.450,-30.880,-42.532,179.836,5.653,149.047
C00735=1192.445,-30.631,-42.545,179.839,5.653,149.047
C00736=1192.440,-30.381,-42.557,179.841,5.654,149.046
C00737=1192.435,-30.131,-42.570,179.844,5.655,149.045
C00738=1192.429,-29.881,-42.583,179.846,5.654,149.045
C00739=1192.424,-29.632,-42.596,179.848,5.655,149.044
C00740=1192.419,-29.383,-42.608,179.850,5.656,149.044
C00741=1192.414,-29.133,-42.620,179.853,5.656,149.043
C00742=1192.409,-28.883,-42.633,179.856,5.656,149.042
C00743=1192.404,-28.634,-42.646,179.858,5.656,149.041
C00744=1192.399,-28.384,-42.658,179.860,5.657,149.041
C00745=1192.394,-28.135,-42.671,179.863,5.657,149.040
C00746=1192.388,-27.884,-42.684,179.865,5.658,149.040
C00747=1192.383,-27.635,-42.696,179.868,5.658,149.039
C00748=1192.378,-27.385,-42.709,179.870,5.658,149.038
C00749=1192.373,-27.136,-42.721,179.872,5.659,149.038
C00750=1192.368,-26.886,-42.734,179.875,5.659,149.037
C00751=1192.363,-26.637,-42.747,179.878,5.660,149.036
C00752=1192.357,-26.387,-42.760,179.880,5.660,149.036
C00753=1192.352,-26.138,-42.773,179.882,5.660,149.035
C00754=1192.348,-25.887,-42.785,179.884,5.661,149.034
C00755=1192.342,-25.638,-42.798,179.887,5.661,149.034
C00756=1192.337,-25.388,-42.810,179.890,5.662,149.033
C00757=1192.332,-25.139,-42.823,179.892,5.662,149.032
C00758=1192.327,-24.889,-42.836,179.895,5.662,149.032
C00759=1192.322,-24.640,-42.849,179.897,5.663,149.031
C00760=1192.317,-24.390,-42.862,179.899,5.663,149.030
C00761=1192.312,-24.140,-42.875,179.902,5.663,149.030
C00762=1192.306,-23.891,-42.888,179.905,5.664,149.029
C00763=1192.301,-23.621,-42.901,179.907,5.664,149.028
C00764=1192.296,-23.352,-42.915,179.910,5.665,149.028
C00765=1192.290,-23.082,-42.929,179.913,5.665,149.027
C00766=1192.285,-22.812,-42.943,179.915,5.665,149.026
C00767=1192.279,-22.562,-42.956,179.917,5.666,149.026
C00768=1192.274,-22.313,-42.969,179.920,5.666,149.025
C00769=1192.269,-22.063,-42.982,179.922,5.667,149.024
C00770=1192.264,-21.813,-42.995,179.925,5.667,149.024
C00771=1192.258,-21.564,-43.007,179.928,5.668,149.023
C00772=1192.253,-21.315,-43.020,179.929,5.668,149.023
C00773=1192.249,-21.065,-43.033,179.932,5.668,149.022
C00774=1192.243,-20.815,-43.046,179.934,5.669,149.021
C00775=1192.238,-20.566,-43.059,179.937,5.669,149.020
C00776=1192.233,-20.316,-43.072,179.940,5.670,149.020
C00777=1192.227,-20.066,-43.085,179.942,5.670,149.019
C00778=1192.223,-19.817,-43.099,179.944,5.670,149.019
C00779=1192.218,-19.567,-43.111,179.947,5.671,149.018
C00780=1192.212,-19.318,-43.124,179.949,5.671,149.017
C00781=1192.208,-19.068,-43.137,179.952,5.672,149.017
C00782=1192.203,-18.819,-43.150,179.954,5.672,149.016
C00783=1192.197,-18.569,-43.163,179.957,5.673,149.015
C00784=1192.192,-18.319,-43.176,179.959,5.672,149.015
C00785=1192.187,-18.070,-43.189,179.962,5.673,149.014
C00786=1192.181,-17.821,-43.203,179.964,5.674,149.014
C00787=1192.177,-17.571,-43.216,179.966,5.674,149.013
C00788=1192.171,-17.321,-43.229,179.969,5.675,149.012
C00789=1192.167,-17.071,-43.242,179.972,5.675,149.011
C00790=1192.161,-16.822,-43.254,179.973,5.675,149.011
C00791=1192.156,-16.572,-43.267,179.976,5.676,149.010
C00792=1192.151,-16.323,-43.281,179.979,5.676,149.010
C00793=1192.146,-16.073,-43.294,179.981,5.677,149.009
C00794=1192.141,-15.823,-43.307,179.984,5.677,149.008
C00795=1192.136,-15.574,-43.320,179.986,5.678,149.008
C00796=1192.130,-15.324,-43.333,179.988,5.678,149.007
C00797=1192.126,-15.075,-43.347,179.991,5.678,149.006
C00798=1192.120,-14.825,-43.360,179.993,5.679,149.006
C00799=1192.115,-14.575,-43.373,179.996,5.679,149.005
C00800=1192.110,-14.325,-43.386,179.998,5.680,149.005
C00801=1192.105,-14.076,-43.400,-179.999,5.680,149.004
C00802=1192.100,-13.827,-43.412,-179.996,5.681,149.003
C00803=1192.094,-13.577,-43.426,-179.994,5.680,149.002
C00804=1192.090,-13.328,-43.439,-179.992,5.681,149.002
C00805=1192.084,-13.078,-43.453,-179.989,5.682,149.001
C00806=1192.080,-12.828,-43.465,-179.987,5.682,149.001
C00807=1192.074,-12.578,-43.479,-179.984,5.683,149.000
C00808=1192.070,-12.329,-43.492,-179.981,5.683,148.999
C00809=1192.064,-12.079,-43.506,-179.979,5.684,148.999
C00810=1192.059,-11.829,-43.519,-179.977,5.684,148.998
C00811=1192.054,-11.580,-43.532,-179.975,5.684,148.997
C00812=1192.049,-11.330,-43.545,-179.972,5.685,148.997
C00813=1192.044,-11.081,-43.559,-179.970,5.686,148.996
C00814=1192.039,-10.831,-43.572,-179.967,5.686,148.996
C00815=1192.033,-10.582,-43.585,-179.964,5.686,148.995
C00816=1192.029,-10.332,-43.599,-179.962,5.687,148.994
C00817=1192.023,-10.082,-43.612,-179.959,5.687,148.993
C00818=1192.019,-9.832,-43.625,-179.958,5.687,148.993
C00819=1192.013,-9.583,-43.639,-179.955,5.688,148.992
C00820=1192.009,-9.333,-43.652,-179.952,5.688,148.992
C00821=1192.003,-9.084,-43.666,-179.950,5.689,148.991
C00822=1191.998,-8.834,-43.680,-179.947,5.690,148.990
C00823=1191.993,-8.585,-43.693,-179.945,5.690,148.990
C00824=1191.988,-8.335,-43.707,-179.942,5.691,148.989
C00825=1191.983,-8.086,-43.719,-179.939,5.691,148.988
C00826=1191.978,-7.836,-43.733,-179.937,5.691,148.988
C00827=1191.972,-7.587,-43.746,-179.935,5.692,148.987
C00828=1191.968,-7.337,-43.760,-179.933,5.692,148.987
C00829=1191.962,-7.087,-43.774,-179.930,5.693,148.986
C00830=1191.957,-6.838,-43.787,-179.927,5.693,148.985
C00831=1191.952,-6.588,-43.800,-179.925,5.694,148.985
C00832=1191.947,-6.339,-43.815,-179.922,5.694,148.984
C00833=1191.942,-6.089,-43.828,-179.920,5.695,148.983
C00834=1191.937,-5.840,-43.842,-179.917,5.695,148.983
C00835=1191.932,-5.590,-43.855,-179.915,5.695,148.982
C00836=1191.926,-5.341,-43.868,-179.913,5.696,148.981
C00837=1191.922,-5.091,-43.883,-179.910,5.696,148.981
C00838=1191.916,-4.842,-43.895,-179.908,5.697,148.980
C00839=1191.911,-4.592,-43.910,-179.905,5.697,148.979
C00840=1191.906,-4.342,-43.923,-179.903,5.698,148.979
C00841=1191.901,-4.093,-43.936,-179.900,5.699,148.978
C00842=1191.896,-3.842,-43.950,-179.897,5.699,148.978
C00843=1191.891,-3.593,-43.964,-179.895,5.700,148.977
C00844=1191.886,-3.344,-43.978,-179.892,5.700,148.976
C00845=1191.881,-3.094,-43.991,-179.891,5.700,148.976
C00846=1191.876,-2.845,-44.005,-179.888,5.701,148.975
C00847=1191.871,-2.595,-44.019,-179.885,5.701,148.974
C00848=1191.865,-2.346,-44.032,-179.883,5.702,148.974
C00849=1191.860,-2.096,-44.046,-179.880,5.702,148.973
C00850=1191.856,-1.846,-44.061,-179.878,5.703,148.972
C00851=1191.850,-1.597,-44.073,-179.875,5.703,148.972
C00852=1191.845,-1.347,-44.087,-179.872,5.704,148.971
C00853=1191.841,-1.098,-44.102,-179.870,5.705,148.971
C00854=1191.835,-0.848,-44.115,-179.868,5.705,148.970
C00855=1191.830,-0.599,-44.129,-179.865,5.706,148.969
C00856=1191.825,-0.350,-44.142,-179.863,5.705,148.969
C00857=1191.820,-0.099,-44.156,-179.860,5.706,148.968
C00858=1191.815,0.151,-44.170,-179.858,5.707,148.967
C00859=1191.809,0.400,-44.184,-179.855,5.707,148.967
C00860=1191.805,0.649,-44.198,-179.853,5.708,148.966
C00861=1191.800,0.899,-44.211,-179.850,5.708,148.965
C00862=1191.794,1.148,-44.225,-179.848,5.709,148.965
C00863=1191.789,1.398,-44.240,-179.845,5.710,148.964
C00864=1191.785,1.647,-44.253,-179.843,5.710,148.964
C00865=1191.779,1.897,-44.267,-179.840,5.710,148.963
C00866=1191.774,2.147,-44.281,-179.838,5.711,148.962
C00867=1191.769,2.416,-44.296,-179.835,5.712,148.962
C00868=1191.763,2.686,-44.311,-179.832,5.712,148.961
C00869=1191.757,2.954,-44.326,-179.830,5.713,148.960
C00870=1191.752,3.223,-44.341,-179.827,5.713,148.960
C00871=1191.747,3.473,-44.355,-179.825,5.714,148.959
C00872=1191.742,3.722,-44.370,-179.822,5.714,148.958
C00873=1191.736,3.972,-44.383,-179.819,5.715,148.958
C00874=1191.732,4.222,-44.397,-179.817,5.716,148.957
C00875=1191.727,4.471,-44.411,-179.814,5.716,148.956
C00876=1191.722,4.720,-44.425,-179.812,5.717,148.956
C00877=1191.717,4.970,-44.439,-179.809,5.717,148.955
C00878=1191.712,5.220,-44.453,-179.807,5.718,148.955
C00879=1191.707,5.469,-44.468,-179.804,5.718,148.954
C00880=1191.701,5.718,-44.481,-179.802,5.718,148.953
C00881=1191.696,5.969,-44.495,-179.800,5.719,148.953
C00882=1191.691,6.218,-44.509,-179.797,5.719,148.952
C00883=1191.687,6.468,-44.523,-179.795,5.720,148.951
C00884=1191.681,6.717,-44.537,-179.792,5.720,148.951
C00885=1191.676,6.967,-44.551,-179.789,5.721,148.950
C00886=1191.671,7.216,-44.565,-179.787,5.721,148.949
C00887=1191.666,7.466,-44.580,-179.785,5.722,148.949
C00888=1191.661,7.715,-44.594,-179.782,5.723,148.948
C00889=1191.656,7.965,-44.608,-179.779,5.723,148.947
C00890=1191.651,8.214,-44.622,-179.777,5.724,148.947
C00891=1191.646,8.464,-44.636,-179.775,5.725,148.946
C00892=1191.641,8.714,-44.651,-179.772,5.725,148.946
C00893=1191.635,8.963,-44.665,-179.769,5.726,148.945
C00894=1191.630,9.213,-44.679,-179.767,5.726,148.944
C00895=1191.625,9.462,-44.693,-179.764,5.727,148.944
C00896=1191.620,9.712,-44.707,-179.762,5.727,148.943
C00897=1191.616,9.962,-44.722,-179.759,5.728,148.942
C00898=1191.610,10.211,-44.736,-179.756,5.728,148.942
C00899=1191.605,10.460,-44.750,-179.754,5.729,148.941
C00900=1191.600,10.710,-44.764,-179.752,5.730,148.941
C00901=1191.595,10.960,-44.779,-179.749,5.730,148.940
C00902=1191.590,11.210,-44.793,-179.746,5.731,148.939
C00903=1191.585,11.458,-44.807,-179.744,5.732,148.939
C00904=1191.580,11.708,-44.822,-179.741,5.732,148.938
C00905=1191.575,11.957,-44.836,-179.739,5.733,148.937
C00906=1191.570,12.207,-44.850,-179.736,5.733,148.937
C00907=1191.565,12.457,-44.865,-179.734,5.734,148.936
C00908=1191.560,12.706,-44.879,-179.731,5.734,148.936
C00909=1191.555,12.955,-44.893,-179.729,5.735,148.935
C00910=1191.550,13.205,-44.907,-179.726,5.735,148.934
C00911=1191.545,13.454,-44.922,-179.725,5.735,148.934
C00912=1191.539,13.704,-44.937,-179.722,5.736,148.933
C00913=1191.534,13.954,-44.951,-179.719,5.736,148.932
C00914=1191.529,14.204,-44.965,-179.717,5.737,148.932
C00915=1191.524,14.453,-44.980,-179.714,5.738,148.931
C00916=1191.519,14.702,-44.994,-179.712,5.738,148.931
C00917=1191.514,14.952,-45.009,-179.709,5.739,148.930
C00918=1191.509,15.201,-45.023,-179.706,5.739,148.929
C00919=1191.504,15.451,-45.037,-179.704,5.740,148.929
C00920=1191.499,15.701,-45.051,-179.702,5.741,148.928
C00921=1191.494,15.950,-45.067,-179.699,5.741,148.927
C00922=1191.489,16.200,-45.081,-179.696,5.742,148.927
C00923=1191.484,16.449,-45.096,-179.694,5.742,148.926
C00924=1191.479,16.699,-45.110,-179.692,5.743,148.926
C00925=1191.474,16.948,-45.124,-179.689,5.743,148.925
C00926=1191.469,17.197,-45.139,-179.686,5.744,148.924
C00927=1191.463,17.447,-45.154,-179.684,5.745,148.924
C00928=1191.459,17.696,-45.169,-179.681,5.745,148.923
C00929=1191.454,17.946,-45.183,-179.679,5.746,148.922
C00930=1191.449,18.196,-45.197,-179.676,5.746,148.922
C00931=1191.444,18.445,-45.212,-179.674,5.747,148.921
C00932=1191.439,18.695,-45.226,-179.671,5.748,148.921
C00933=1191.433,18.945,-45.241,-179.668,5.749,148.920
C00934=1191.429,19.194,-45.256,-179.665,5.749,148.919
C00935=1191.424,19.443,-45.271,-179.663,5.750,148.919
C00936=1191.419,19.693,-45.285,-179.661,5.751,148.918
C00937=1191.413,19.943,-45.300,-179.658,5.751,148.917
C00938=1191.408,20.192,-45.315,-179.655,5.752,148.917
C00939=1191.403,20.442,-45.329,-179.653,5.753,148.916
C00940=1191.399,20.691,-45.344,-179.651,5.753,148.916
C00941=1191.393,20.941,-45.359,-179.648,5.754,148.915
C00942=1191.388,21.190,-45.374,-179.646,5.755,148.914
C00943=1191.384,21.440,-45.388,-179.643,5.755,148.914
C00944=1191.378,21.688,-45.403,-179.640,5.756,148.913
C00945=1191.373,21.938,-45.418,-179.638,5.756,148.912
C00946=1191.368,22.188,-45.432,-179.636,5.757,148.912
C00947=1191.363,22.437,-45.447,-179.633,5.757,148.911
C00948=1191.357,22.687,-45.462,-179.630,5.758,148.911
C00949=1191.353,22.936,-45.477,-179.628,5.758,148.910
C00950=1191.348,23.186,-45.491,-179.626,5.759,148.909
C00951=1191.343,23.435,-45.506,-179.623,5.760,148.909
C00952=1191.337,23.685,-45.521,-179.620,5.760,148.908
C00953=1191.333,23.935,-45.536,-179.618,5.761,148.907
C00954=1191.328,24.185,-45.551,-179.615,5.762,148.907
C00955=1191.323,24.434,-45.566,-179.613,5.762,148.906
C00956=1191.318,24.684,-45.580,-179.610,5.763,148.906
C00957=1191.313,24.933,-45.595,-179.608,5.764,148.905
C00958=1191.308,25.182,-45.611,-179.605,5.764,148.904
C00959=1191.303,25.432,-45.625,-179.603,5.765,148.904
C00960=1191.298,25.681,-45.641,-179.600,5.765,148.903
C00961=1191.293,25.931,-45.655,-179.598,5.766,148.903
C00962=1191.288,26.180,-45.670,-179.595,5.766,148.902
C00963=1191.282,26.430,-45.685,-179.592,5.768,148.901
C00964=1191.278,26.679,-45.700,-179.589,5.768,148.901
C00965=1191.273,26.928,-45.715,-179.587,5.769,148.900
C00966=1191.267,27.178,-45.730,-179.585,5.770,148.900
C00967=1191.263,27.427,-45.745,-179.582,5.770,148.899
C00968=1191.257,27.677,-45.760,-179.580,5.771,148.898
C00969=1191.252,27.926,-45.775,-179.577,5.772,148.898
C00970=1191.247,28.176,-45.790,-179.574,5.772,148.897
C00971=1191.242,28.445,-45.806,-179.572,5.773,148.896
C00972=1191.236,28.714,-45.822,-179.569,5.773,148.896
C00973=1191.231,28.982,-45.839,-179.566,5.774,148.895
C00974=1191.225,29.251,-45.855,-179.563,5.775,148.894
C00975=1191.221,29.501,-45.870,-179.561,5.776,148.894
C00976=1191.216,29.751,-45.885,-179.558,5.776,148.893
C00977=1191.211,30.000,-45.900,-179.556,5.777,148.893
C00978=1191.206,30.249,-45.915,-179.554,5.778,148.892
C00979=1191.201,30.498,-45.931,-179.551,5.778,148.891
C00980=1191.196,30.748,-45.945,-179.548,5.779,148.891
C00981=1191.191,30.998,-45.961,-179.546,5.779,148.890
C00982=1191.186,31.247,-45.976,-179.544,5.780,148.890
C00983=1191.181,31.497,-45.992,-179.540,5.781,148.889
C00984=1191.176,31.746,-46.006,-179.538,5.782,148.888
C00985=1191.171,31.996,-46.022,-179.536,5.783,148.888
C00986=1191.165,32.245,-46.037,-179.533,5.783,148.887
C00987=1191.161,32.494,-46.052,-179.530,5.784,148.886
C00988=1191.155,32.744,-46.068,-179.528,5.784,148.886
C00989=1191.150,32.993,-46.082,-179.525,5.785,148.885
C00990=1191.146,33.244,-46.098,-179.523,5.786,148.885
C00991=1191.141,33.493,-46.113,-179.520,5.786,148.884
C00992=1191.136,33.742,-46.128,-179.518,5.787,148.883
C00993=1191.131,33.991,-46.143,-179.515,5.788,148.883
C00994=1191.126,34.241,-46.159,-179.512,5.789,148.882
C00995=1191.121,34.491,-46.175,-179.510,5.790,148.882
C00996=1191.116,34.740,-46.189,-179.507,5.790,148.881
C00997=1191.110,34.990,-46.205,-179.505,5.791,148.880
C00998=1191.106,35.239,-46.220,-179.502,5.791,148.880
C00999=1191.100,35.488,-46.235,-179.500,5.792,148.879
C01000=1191.095,35.738,-46.251,-179.497,5.793,148.879
C01001=1191.091,35.987,-46.266,-179.495,5.793,148.878
C01002=1191.086,36.237,-46.282,-179.492,5.794,148.877
C01003=1191.081,36.486,-46.297,-179.490,5.795,148.877
C01004=1191.075,36.735,-46.313,-179.487,5.796,148.876
C01005=1191.071,36.985,-46.329,-179.484,5.797,148.876
C01006=1191.066,37.235,-46.344,-179.482,5.797,148.875
C01007=1191.061,37.484,-46.359,-179.479,5.798,148.874
C01008=1191.055,37.733,-46.375,-179.477,5.798,148.874
C01009=1191.051,37.982,-46.390,-179.474,5.799,148.873
C01010=1191.046,38.233,-46.406,-179.472,5.800,148.872
C01011=1191.040,38.482,-46.421,-179.469,5.800,148.872
C01012=1191.036,38.731,-46.436,-179.467,5.801,148.871
C01013=1191.030,38.980,-46.452,-179.464,5.802,148.871
C01014=1191.026,39.231,-46.468,-179.461,5.803,148.870
C01015=1191.021,39.480,-46.483,-179.459,5.804,148.870
C01016=1191.016,39.729,-46.498,-179.456,5.804,148.869
C01017=1191.011,39.979,-46.514,-179.454,5.805,148.868
C01018=1191.005,40.229,-46.530,-179.451,5.806,148.868
C01019=1191.001,40.478,-46.545,-179.449,5.806,148.867
C01020=1190.995,40.727,-46.560,-179.446,5.807,148.866
C01021=1190.991,40.977,-46.576,-179.443,5.808,148.866
C01022=1190.985,41.227,-46.592,-179.441,5.809,148.865
C01023=1190.981,41.476,-46.607,-179.438,5.810,148.865
C01024=1190.976,41.725,-46.624,-179.436,5.810,148.864
C01025=1190.971,41.975,-46.639,-179.433,5.811,148.864
C01026=1190.965,42.224,-46.655,-179.431,5.811,148.863
C01027=1190.961,42.473,-46.670,-179.428,5.812,148.862
C01028=1190.956,42.723,-46.686,-179.425,5.814,148.862
C01029=1190.950,42.973,-46.701,-179.423,5.814,148.861
C01030=1190.945,43.221,-46.718,-179.420,5.815,148.860
C01031=1190.941,43.471,-46.734,-179.418,5.816,148.860
C01032=1190.936,43.721,-46.749,-179.415,5.816,148.859
C01033=1190.931,43.970,-46.764,-179.413,5.817,148.859
C01034=1190.926,44.220,-46.780,-179.410,5.817,148.858
C01035=1190.921,44.469,-46.796,-179.407,5.819,148.858
C01036=1190.915,44.718,-46.812,-179.405,5.819,148.857
C01037=1190.911,44.968,-46.828,-179.402,5.820,148.856
C01038=1190.906,45.217,-46.843,-179.400,5.821,148.856
C01039=1190.901,45.467,-46.859,-179.397,5.821,148.855
C01040=1190.896,45.716,-46.875,-179.395,5.822,148.855
C01041=1190.891,45.966,-46.891,-179.392,5.823,148.854
C01042=1190.886,46.216,-46.907,-179.389,5.824,148.853
C01043=1190.881,46.465,-46.923,-179.387,5.825,148.853
C01044=1190.875,46.714,-46.939,-179.384,5.825,148.852
C01045=1190.871,46.964,-46.954,-179.382,5.826,148.851
C01046=1190.866,47.213,-46.970,-179.380,5.827,148.851
C01047=1190.861,47.463,-46.986,-179.377,5.827,148.850
C01048=1190.856,47.712,-47.002,-179.374,5.829,148.850
C01049=1190.851,47.961,-47.018,-179.372,5.830,148.849
C01050=1190.846,48.211,-47.034,-179.369,5.830,148.849
C01051=1190.841,48.460,-47.050,-179.366,5.831,148.848
C01052=1190.836,48.710,-47.066,-179.364,5.831,148.847
C01053=1190.831,48.959,-47.082,-179.361,5.833,148.847
C01054=1190.826,49.209,-47.098,-179.358,5.833,148.846
C01055=1190.821,49.458,-47.114,-179.356,5.834,148.846
C01056=1190.816,49.708,-47.130,-179.354,5.835,148.845
C01057=1190.812,49.957,-47.146,-179.351,5.835,148.844
C01058=1190.807,50.206,-47.162,-179.349,5.836,148.844
C01059=1190.802,50.456,-47.177,-179.346,5.838,148.843
C01060=1190.797,50.705,-47.194,-179.343,5.838,148.843
C01061=1190.792,50.955,-47.210,-179.341,5.839,148.842
C01062=1190.787,51.204,-47.226,-179.338,5.839,148.841
C01063=1190.781,51.453,-47.242,-179.335,5.840,148.841
C01064=1190.777,51.703,-47.258,-179.333,5.842,148.840
C01065=1190.772,51.952,-47.274,-179.330,5.842,148.840
C01066=1190.767,52.202,-47.291,-179.327,5.843,148.839
C01067=1190.762,52.451,-47.306,-179.325,5.844,148.839
C01068=1190.757,52.701,-47.323,-179.323,5.844,148.838
C01069=1190.752,52.950,-47.338,-179.319,5.845,148.837
C01070=1190.747,53.199,-47.355,-179.317,5.846,148.837
C01071=1190.741,53.449,-47.371,-179.315,5.847,148.836
C01072=1190.737,53.699,-47.388,-179.312,5.847,148.835
C01073=1190.732,53.947,-47.404,-179.310,5.848,148.835
C01074=1190.727,54.198,-47.420,-179.307,5.850,148.834
C01075=1190.721,54.466,-47.437,-179.304,5.850,148.834
C01076=1190.716,54.734,-47.455,-179.301,5.851,148.833
C01077=1190.711,55.003,-47.472,-179.299,5.852,148.833
C01078=1190.706,55.271,-47.490,-179.296,5.853,148.832
C01079=1190.701,55.521,-47.506,-179.293,5.853,148.831
C01080=1190.696,55.770,-47.522,-179.291,5.854,148.831
C01081=1190.691,56.020,-47.539,-179.288,5.856,148.830
C01082=1190.685,56.269,-47.555,-179.285,5.856,148.830
C01083=1190.681,56.518,-47.572,-179.283,5.857,148.829
C01084=1190.676,56.768,-47.587,-179.281,5.858,148.828
C01085=1190.671,57.017,-47.604,-179.277,5.859,148.828
C01086=1190.666,57.266,-47.620,-179.275,5.860,148.827
C01087=1190.661,57.516,-47.636,-179.273,5.860,148.827
C01088=1190.655,57.765,-47.653,-179.270,5.861,148.826
C01089=1190.651,58.015,-47.670,-179.268,5.862,148.826
C01090=1190.646,58.264,-47.687,-179.265,5.863,148.825
C01091=1190.641,58.514,-47.702,-179.262,5.864,148.824
C01092=1190.637,58.763,-47.719,-179.260,5.865,148.824
C01093=1190.631,59.012,-47.735,-179.257,5.865,148.823
C01094=1190.626,59.262,-47.752,-179.254,5.867,148.823
C01095=1190.621,59.511,-47.768,-179.252,5.867,148.822
C01096=1190.616,59.761,-47.785,-179.249,5.868,148.821
C01097=1190.612,60.010,-47.801,-179.247,5.869,148.821
C01098=1190.606,60.259,-47.818,-179.244,5.870,148.820
C01099=1190.601,60.509,-47.834,-179.242,5.871,148.820
C01100=1190.596,60.758,-47.850,-179.239,5.872,148.819
C01101=1190.592,61.008,-47.867,-179.236,5.872,148.818
C01102=1190.587,61.257,-47.884,-179.234,5.874,148.818
C01103=1190.581,61.506,-47.901,-179.231,5.874,148.817
C01104=1190.577,61.756,-47.917,-179.228,5.875,148.817
C01105=1190.572,62.006,-47.933,-179.226,5.876,148.816
C01106=1190.567,62.255,-47.950,-179.223,5.877,148.816
C01107=1190.562,62.504,-47.967,-179.221,5.878,148.815
C01108=1190.557,62.754,-47.984,-179.218,5.879,148.815
C01109=1190.552,63.003,-48.000,-179.216,5.879,148.814
C01110=1190.547,63.252,-48.017,-179.213,5.881,148.813
C01111=1190.542,63.501,-48.033,-179.210,5.881,148.813
C01112=1190.538,63.751,-48.050,-179.208,5.882,148.812
C01113=1190.532,64.001,-48.067,-179.206,5.883,148.812
C01114=1190.527,64.250,-48.083,-179.202,5.884,148.811
C01115=1190.522,64.499,-48.100,-179.200,5.885,148.811
C01116=1190.517,64.749,-48.117,-179.198,5.886,148.810
C01117=1190.512,64.998,-48.133,-179.195,5.886,148.809
C01118=1190.508,65.247,-48.150,-179.192,5.888,148.809
C01119=1190.502,65.497,-48.167,-179.190,5.888,148.808
C01120=1190.498,65.747,-48.184,-179.187,5.889,148.808
C01121=1190.493,65.995,-48.200,-179.185,5.890,148.807
C01122=1190.488,66.245,-48.217,-179.182,5.891,148.807
C01123=1190.483,66.495,-48.234,-179.179,5.892,148.806
C01124=1190.478,66.744,-48.250,-179.177,5.893,148.805
C01125=1190.473,66.993,-48.268,-179.174,5.894,148.805
C01126=1190.468,67.243,-48.284,-179.171,5.895,148.804
C01127=1190.463,67.493,-48.302,-179.169,5.896,148.804
C01128=1190.458,67.741,-48.318,-179.167,5.896,148.803
C01129=1190.454,67.991,-48.335,-179.163,5.898,148.802
C01130=1190.449,68.240,-48.353,-179.161,5.898,148.802
C01131=1190.444,68.490,-48.369,-179.159,5.899,148.801
C01132=1190.438,68.739,-48.386,-179.156,5.901,148.801
C01133=1190.434,68.988,-48.403,-179.153,5.901,148.800
C01134=1190.429,69.238,-48.419,-179.151,5.902,148.800
C01135=1190.424,69.487,-48.437,-179.149,5.903,148.799
C01136=1190.419,69.736,-48.453,-179.145,5.904,148.799
C01137=1190.414,69.986,-48.470,-179.143,5.905,148.798
C01138=1190.409,70.235,-48.487,-179.141,5.906,148.797
C01139=1190.405,70.485,-48.505,-179.137,5.907,148.797
C01140=1190.400,70.733,-48.521,-179.135,5.908,148.796
C01141=1190.394,70.983,-48.538,-179.133,5.908,148.796
C01142=1190.390,71.233,-48.555,-179.130,5.910,148.795
C01143=1190.385,71.482,-48.572,-179.127,5.911,148.795
C01144=1190.380,71.731,-48.589,-179.125,5.911,148.794
C01145=1190.375,71.980,-48.607,-179.122,5.912,148.794
C01146=1190.370,72.230,-48.623,-179.119,5.913,148.793
C01147=1190.365,72.480,-48.641,-179.117,5.914,148.792
C01148=1190.360,72.729,-48.657,-179.114,5.915,148.792
C01149=1190.356,72.978,-48.675,-179.112,5.917,148.791
C01150=1190.350,73.227,-48.692,-179.109,5.917,148.791
C01151=1190.345,73.477,-48.709,-179.107,5.918,148.790
C01152=1190.340,73.726,-48.727,-179.104,5.919,148.790
C01153=1190.336,73.976,-48.743,-179.101,5.920,148.789
C01154=1190.331,74.225,-48.761,-179.099,5.921,148.789
C01155=1190.326,74.474,-48.777,-179.096,5.922,148.788
C01156=1190.321,74.723,-48.795,-179.094,5.923,148.787
C01157=1190.315,74.973,-48.812,-179.091,5.924,148.787
C01158=1190.311,75.223,-48.829,-179.088,5.925,148.786
C01159=1190.306,75.472,-48.847,-179.086,5.926,148.786
C01160=1190.302,75.721,-48.864,-179.083,5.926,148.785
C01161=1190.296,75.971,-48.881,-179.080,5.928,148.785
C01162=1190.291,76.220,-48.898,-179.078,5.929,148.784
C01163=1190.286,76.469,-48.915,-179.076,5.930,148.784
C01164=1190.281,76.718,-48.933,-179.072,5.931,148.783
C01165=1190.277,76.968,-48.950,-179.070,5.932,148.782
C01166=1190.272,77.218,-48.967,-179.068,5.932,148.782
C01167=1190.267,77.467,-48.985,-179.065,5.934,148.781
C01168=1190.262,77.716,-49.002,-179.062,5.935,148.781
C01169=1190.257,77.965,-49.020,-179.060,5.935,148.780
C01170=1190.252,78.215,-49.037,-179.057,5.937,148.780
C01171=1190.247,78.463,-49.054,-179.054,5.937,148.779
C01172=1190.242,78.713,-49.071,-179.052,5.938,148.779
C01173=1190.237,78.962,-49.089,-179.049,5.940,148.778
C01174=1190.232,79.212,-49.106,-179.047,5.941,148.777
C01175=1190.228,79.461,-49.124,-179.044,5.941,148.777
C01176=1190.223,79.711,-49.141,-179.041,5.943,148.776
C01177=1190.218,79.960,-49.159,-179.039,5.943,148.776
C01178=1190.213,80.209,-49.176,-179.036,5.945,148.775
C01179=1190.208,80.478,-49.195,-179.033,5.946,148.775
C01180=1190.202,80.746,-49.214,-179.030,5.947,148.774
C01181=1190.197,81.015,-49.232,-179.028,5.948,148.773
C01182=1190.192,81.283,-49.252,-179.025,5.949,148.773
C01183=1190.186,81.533,-49.269,-179.022,5.950,148.772
C01184=1190.182,81.782,-49.286,-179.020,5.950,148.772
C01185=1190.177,82.031,-49.304,-179.017,5.952,148.771
C01186=1190.172,82.281,-49.322,-179.014,5.953,148.771
C01187=1190.167,82.530,-49.339,-179.012,5.954,148.770
C01188=1190.163,82.779,-49.356,-179.009,5.955,148.769
C01189=1190.158,83.028,-49.374,-179.007,5.956,148.769
C01190=1190.153,83.278,-49.392,-179.004,5.957,148.768
C01191=1190.148,83.527,-49.409,-179.001,5.958,148.768
C01192=1190.143,83.777,-49.427,-178.999,5.959,148.767
C01193=1190.138,84.026,-49.445,-178.996,5.960,148.767
C01194=1190.133,84.275,-49.462,-178.994,5.961,148.766
C01195=1190.129,84.524,-49.480,-178.991,5.963,148.766
C01196=1190.124,84.774,-49.498,-178.988,5.963,148.765
C01197=1190.118,85.023,-49.515,-178.986,5.964,148.765
C01198=1190.114,85.273,-49.533,-178.983,5.966,148.764
C01199=1190.109,85.522,-49.551,-178.981,5.966,148.764
C01200=1190.104,85.771,-49.569,-178.977,5.968,148.763
C01201=1190.099,86.020,-49.586,-178.975,5.969,148.763
C01202=1190.094,86.270,-49.604,-178.973,5.969,148.762
C01203=1190.089,86.519,-49.622,-178.970,5.971,148.762
C01204=1190.084,86.768,-49.640,-178.967,5.972,148.761
C01205=1190.079,87.018,-49.657,-178.965,5.972,148.760
C01206=1190.074,87.267,-49.675,-178.962,5.974,148.760
C01207=1190.069,87.516,-49.693,-178.959,5.974,148.759
C01208=1190.065,87.765,-49.711,-178.957,5.976,148.759
C01209=1190.060,88.014,-49.729,-178.954,5.977,148.758
C01210=1190.054,88.264,-49.746,-178.951,5.978,148.758
C01211=1190.049,88.513,-49.764,-178.949,5.979,148.757
C01212=1190.045,88.763,-49.783,-178.947,5.980,148.757
C01213=1190.040,89.012,-49.801,-178.943,5.981,148.756
C01214=1190.036,89.261,-49.818,-178.941,5.982,148.756
C01215=1190.031,89.510,-49.836,-178.938,5.984,148.755
C01216=1190.026,89.760,-49.854,-178.936,5.984,148.754
C01217=1190.021,90.009,-49.871,-178.933,5.985,148.754
C01218=1190.016,90.259,-49.889,-178.931,5.987,148.753
C01219=1190.011,90.508,-49.907,-178.928,5.987,148.753
C01220=1190.006,90.757,-49.925,-178.925,5.989,148.752
C01221=1190.001,91.006,-49.943,-178.923,5.990,148.752
C01222=1189.997,91.256,-49.961,-178.920,5.991,148.751
C01223=1189.992,91.505,-49.979,-178.917,5.992,148.751
C01224=1189.987,91.755,-49.998,-178.915,5.993,148.750
C01225=1189.982,92.004,-50.016,-178.912,5.995,148.750
C01226=1189.977,92.253,-50.034,-178.910,5.995,148.749
C01227=1189.972,92.502,-50.052,-178.907,5.997,148.749
C01228=1189.967,92.751,-50.070,-178.905,5.997,148.748
C01229=1189.963,93.001,-50.088,-178.902,5.999,148.748
C01230=1189.958,93.250,-50.106,-178.899,6.000,148.747
C01231=1189.953,93.500,-50.124,-178.897,6.001,148.747
C01232=1189.948,93.749,-50.142,-178.894,6.002,148.746
C01233=1189.943,93.998,-50.160,-178.892,6.003,148.746
C01234=1189.938,94.247,-50.178,-178.889,6.004,148.745
C01235=1189.934,94.497,-50.196,-178.886,6.005,148.744
C01236=1189.929,94.746,-50.214,-178.883,6.007,148.744
C01237=1189.923,94.996,-50.233,-178.881,6.007,148.743
C01238=1189.918,95.245,-50.251,-178.878,6.009,148.743
C01239=1189.914,95.493,-50.270,-178.876,6.010,148.742
C01240=1189.909,95.743,-50.288,-178.873,6.010,148.742
C01241=1189.904,95.992,-50.306,-178.870,6.012,148.741
C01242=1189.899,96.242,-50.324,-178.868,6.013,148.741
C01243=1189.895,96.491,-50.342,-178.865,6.014,148.740
C01244=1189.889,96.740,-50.361,-178.862,6.015,148.740
C01245=1189.885,96.990,-50.379,-178.860,6.017,148.739
C01246=1189.880,97.239,-50.398,-178.858,6.018,148.739
C01247=1189.875,97.488,-50.416,-178.854,6.019,148.738
C01248=1189.870,97.737,-50.434,-178.852,6.020,148.738
C01249=1189.866,97.987,-50.452,-178.849,6.021,148.737
C01250=1189.860,98.236,-50.470,-178.847,6.022,148.737
C01251=1189.856,98.485,-50.489,-178.844,6.024,148.736
C01252=1189.851,98.734,-50.507,-178.842,6.024,148.736
C01253=1189.846,98.984,-50.526,-178.839,6.025,148.735
C01254=1189.841,99.234,-50.544,-178.836,6.027,148.735
C01255=1189.836,99.482,-50.563,-178.834,6.027,148.734
C01256=1189.831,99.731,-50.581,-178.831,6.029,148.733
C01257=1189.827,99.981,-50.599,-178.829,6.030,148.733
C01258=1189.821,100.231,-50.618,-178.826,6.031,148.732
C01259=1189.817,100.479,-50.636,-178.824,6.032,148.732
C01260=1189.812,100.728,-50.654,-178.820,6.034,148.731
C01261=1189.807,100.978,-50.673,-178.818,6.035,148.731
C01262=1189.802,101.227,-50.692,-178.815,6.036,148.730
C01263=1189.797,101.476,-50.710,-178.813,6.037,148.730
C01264=1189.793,101.726,-50.728,-178.810,6.038,148.729
C01265=1189.788,101.975,-50.748,-178.808,6.039,148.729
C01266=1189.783,102.224,-50.766,-178.805,6.041,148.728
C01267=1189.778,102.474,-50.784,-178.802,6.041,148.728
C01268=1189.773,102.723,-50.803,-178.799,6.043,148.727
C01269=1189.768,102.972,-50.821,-178.797,6.044,148.727
C01270=1189.764,103.221,-50.840,-178.794,6.046,148.726
C01271=1189.758,103.471,-50.859,-178.792,6.046,148.726
C01272=1189.753,103.720,-50.877,-178.789,6.048,148.725
C01273=1189.749,103.969,-50.896,-178.787,6.049,148.725
C01274=1189.744,104.219,-50.914,-178.784,6.050,148.724
C01275=1189.739,104.467,-50.933,-178.781,6.051,148.724
C01276=1189.735,104.717,-50.952,-178.778,6.052,148.723
C01277=1189.730,104.966,-50.971,-178.776,6.053,148.723
C01278=1189.725,105.215,-50.989,-178.773,6.055,148.722
C01279=1189.720,105.465,-51.008,-178.771,6.056,148.722
C01280=1189.715,105.714,-51.026,-178.768,6.057,148.721
C01281=1189.710,105.963,-51.045,-178.765,6.058,148.721
C01282=1189.705,106.213,-51.064,-178.763,6.060,148.720
C01283=1189.701,106.480,-51.084,-178.760,6.061,148.720
C01284=1189.695,106.749,-51.104,-178.757,6.062,148.719
C01285=1189.689,107.018,-51.125,-178.754,6.063,148.719
C01286=1189.685,107.286,-51.145,-178.751,6.065,148.718
C01287=1189.680,107.535,-51.164,-178.749,6.066,148.718
C01288=1189.675,107.785,-51.182,-178.746,6.067,148.717
C01289=1189.670,108.033,-51.202,-178.744,6.068,148.716
C01290=1189.665,108.283,-51.220,-178.741,6.070,148.716
C01291=1189.660,108.532,-51.239,-178.738,6.070,148.715
C01292=1189.656,108.781,-51.258,-178.736,6.072,148.715
C01293=1189.650,109.031,-51.277,-178.733,6.073,148.714
C01294=1189.646,109.280,-51.296,-178.730,6.074,148.714
C01295=1189.641,109.530,-51.315,-178.728,6.076,148.714
C01296=1189.636,109.778,-51.333,-178.725,6.077,148.713
C01297=1189.631,110.028,-51.353,-178.722,6.078,148.713
C01298=1189.627,110.276,-51.372,-178.720,6.079,148.712
C01299=1189.622,110.527,-51.390,-178.717,6.081,148.711
C01300=1189.617,110.775,-51.409,-178.715,6.082,148.711
C01301=1189.612,111.025,-51.429,-178.712,6.083,148.710
C01302=1189.607,111.274,-51.447,-178.709,6.084,148.710
C01303=1189.603,111.523,-51.466,-178.707,6.086,148.710
C01304=1189.597,111.772,-51.486,-178.704,6.086,148.709
C01305=1189.593,112.022,-51.505,-178.701,6.088,148.709
C01306=1189.588,112.271,-51.523,-178.698,6.089,148.708
C01307=1189.584,112.520,-51.542,-178.696,6.090,148.708
C01308=1189.578,112.769,-51.562,-178.693,6.092,148.707
C01309=1189.574,113.018,-51.581,-178.691,6.093,148.706
C01310=1189.569,113.268,-51.599,-178.688,6.094,148.706
C01311=1189.564,113.517,-51.619,-178.685,6.095,148.705
C01312=1189.559,113.766,-51.638,-178.683,6.097,148.705
C01313=1189.555,114.016,-51.657,-178.680,6.099,148.705
C01314=1189.549,114.264,-51.677,-178.677,6.099,148.704
C01315=1189.545,114.514,-51.696,-178.675,6.101,148.704
C01316=1189.540,114.763,-51.714,-178.673,6.102,148.703
C01317=1189.535,115.013,-51.734,-178.669,6.103,148.703
C01318=1189.530,115.261,-51.753,-178.667,6.104,148.702
C01319=1189.526,115.511,-51.772,-178.665,6.106,148.702
C01320=1189.520,115.760,-51.792,-178.661,6.107,148.701
C01321=1189.516,116.009,-51.811,-178.659,6.108,148.701
C01322=1189.511,116.258,-51.830,-178.656,6.110,148.700
C01323=1189.506,116.507,-51.850,-178.654,6.111,148.700
C01324=1189.502,116.756,-51.868,-178.651,6.112,148.699
C01325=1189.497,117.006,-51.888,-178.648,6.114,148.699
C01326=1189.492,117.255,-51.908,-178.646,6.115,148.698
C01327=1189.487,117.504,-51.927,-178.643,6.116,148.698
C01328=1189.483,117.753,-51.946,-178.641,6.117,148.697
C01329=1189.477,118.002,-51.965,-178.638,6.119,148.697
C01330=1189.473,118.252,-51.985,-178.636,6.120,148.696
C01331=1189.468,118.501,-52.005,-178.633,6.121,148.696
C01332=1189.463,118.750,-52.023,-178.630,6.123,148.695
C01333=1189.459,118.999,-52.043,-178.628,6.124,148.695
C01334=1189.453,119.248,-52.062,-178.625,6.125,148.694
C01335=1189.448,119.498,-52.082,-178.623,6.126,148.694
C01336=1189.444,119.747,-52.102,-178.619,6.127,148.693
C01337=1189.439,119.996,-52.120,-178.617,6.129,148.693
C01338=1189.434,120.246,-52.140,-178.615,6.130,148.692
C01339=1189.429,120.494,-52.159,-178.611,6.131,148.692
C01340=1189.424,120.744,-52.179,-178.609,6.133,148.691
C01341=1189.419,120.994,-52.199,-178.607,6.134,148.691
C01342=1189.415,121.242,-52.217,-178.603,6.136,148.690
C01343=1189.410,121.492,-52.237,-178.601,6.136,148.690
C01344=1189.406,121.741,-52.257,-178.598,6.138,148.690
C01345=1189.400,121.989,-52.277,-178.595,6.140,148.689
C01346=1189.396,122.239,-52.296,-178.593,6.141,148.689
C01347=1189.391,122.489,-52.316,-178.590,6.142,148.688
C01348=1189.386,122.737,-52.335,-178.588,6.143,148.688
C01349=1189.382,122.987,-52.354,-178.585,6.145,148.687
C01350=1189.377,123.236,-52.375,-178.582,6.146,148.687
C01351=1189.372,123.485,-52.394,-178.580,6.147,148.686
C01352=1189.367,123.734,-52.414,-178.577,6.149,148.686
C01353=1189.362,123.984,-52.433,-178.574,6.151,148.685
C01354=1189.357,124.232,-52.453,-178.572,6.151,148.685
C01355=1189.352,124.482,-52.473,-178.569,6.153,148.684
C01356=1189.348,124.731,-52.492,-178.566,6.155,148.684
C01357=1189.343,124.981,-52.512,-178.564,6.156,148.684
C01358=1189.338,125.229,-52.532,-178.561,6.157,148.683
C01359=1189.333,125.478,-52.552,-178.559,6.158,148.682
C01360=1189.329,125.728,-52.571,-178.556,6.160,148.682
C01361=1189.325,125.977,-52.591,-178.553,6.161,148.681
C01362=1189.319,126.226,-52.611,-178.551,6.162,148.681
C01363=1189.315,126.475,-52.630,-178.548,6.164,148.681
C01364=1189.310,126.724,-52.651,-178.545,6.165,148.680
C01365=1189.305,126.973,-52.670,-178.543,6.166,148.680
C01366=1189.300,127.223,-52.689,-178.540,6.168,148.679
C01367=1189.296,127.471,-52.710,-178.538,6.170,148.679
C01368=1189.291,127.721,-52.730,-178.535,6.170,148.678
C01369=1189.286,127.971,-52.749,-178.532,6.172,148.678
C01370=1189.281,128.219,-52.769,-178.530,6.174,148.677
C01371=1189.276,128.468,-52.789,-178.527,6.174,148.677
C01372=1189.272,128.717,-52.809,-178.524,6.176,148.676
C01373=1189.267,128.967,-52.829,-178.522,6.178,148.676
C01374=1189.262,129.215,-52.849,-178.520,6.179,148.676
C01375=1189.257,129.465,-52.869,-178.516,6.180,148.675
C01376=1189.252,129.714,-52.889,-178.514,6.182,148.675
C01377=1189.248,129.964,-52.909,-178.512,6.183,148.674
C01378=1189.243,130.213,-52.929,-178.508,6.184,148.674
C01379=1189.238,130.461,-52.949,-178.506,6.186,148.673
C01380=1189.233,130.711,-52.968,-178.504,6.187,148.673
C01381=1189.229,130.960,-52.989,-178.501,6.189,148.672
C01382=1189.224,131.209,-53.009,-178.498,6.190,148.672
C01383=1189.219,131.458,-53.029,-178.496,6.191,148.671
C01384=1189.215,131.707,-53.049,-178.493,6.193,148.671
C01385=1189.209,131.957,-53.069,-178.490,6.194,148.670
C01386=1189.204,132.205,-53.090,-178.488,6.195,148.670
C01387=1189.200,132.474,-53.111,-178.485,6.197,148.670
C01388=1189.194,132.743,-53.132,-178.482,6.198,148.669
C01389=1189.189,133.011,-53.154,-178.479,6.200,148.669
C01390=1189.184,133.280,-53.176,-178.476,6.201,148.668
C01391=1189.179,133.529,-53.196,-178.473,6.203,148.668
C01392=1189.175,133.778,-53.216,-178.471,6.204,148.667
C01393=1189.170,134.028,-53.236,-178.468,6.206,148.667
C01394=1189.165,134.277,-53.257,-178.465,6.207,148.666
C01395=1189.160,134.526,-53.277,-178.462,6.209,148.666
C01396=1189.156,134.775,-53.297,-178.460,6.210,148.665
C01397=1189.151,135.024,-53.318,-178.458,6.212,148.665
C01398=1189.146,135.273,-53.338,-178.454,6.213,148.664
C01399=1189.141,135.522,-53.358,-178.452,6.214,148.664
C01400=1189.136,135.771,-53.378,-178.450,6.216,148.664
C01401=1189.132,136.020,-53.399,-178.447,6.218,148.663
C01402=1189.127,136.270,-53.418,-178.444,6.219,148.663
C01403=1189.122,136.519,-53.439,-178.442,6.220,148.662
C01404=1189.118,136.768,-53.460,-178.439,6.222,148.662
C01405=1189.113,137.017,-53.480,-178.436,6.224,148.661
C01406=1189.108,137.267,-53.500,-178.434,6.224,148.661
C01407=1189.103,137.516,-53.521,-178.431,6.226,148.660
C01408=1189.099,137.765,-53.541,-178.428,6.228,148.660
C01409=1189.094,138.014,-53.561,-178.426,6.229,148.660
C01410=1189.089,138.263,-53.582,-178.423,6.230,148.659
C01411=1189.084,138.511,-53.602,-178.420,6.232,148.659
C01412=1189.079,138.761,-53.622,-178.418,6.234,148.658
C01413=1189.074,139.010,-53.643,-178.415,6.235,148.658
C01414=1189.070,139.259,-53.663,-178.413,6.236,148.657
C01415=1189.065,139.508,-53.684,-178.410,6.238,148.657
C01416=1189.060,139.757,-53.705,-178.407,6.239,148.656
C01417=1189.056,140.006,-53.725,-178.405,6.240,148.656
C01418=1189.051,140.255,-53.745,-178.402,6.242,148.656
C01419=1189.046,140.504,-53.766,-178.399,6.244,148.655
C01420=1189.041,140.754,-53.786,-178.396,6.245,148.655
C01421=1189.037,141.003,-53.806,-178.394,6.246,148.654
C01422=1189.032,141.252,-53.827,-178.392,6.248,148.654
C01423=1189.027,141.501,-53.848,-178.389,6.250,148.654
C01424=1189.022,141.750,-53.869,-178.386,6.251,148.653
C01425=1189.018,141.999,-53.889,-178.384,6.252,148.653
C01426=1189.013,142.248,-53.909,-178.381,6.254,148.652
C01427=1189.008,142.498,-53.930,-178.378,6.256,148.652
C01428=1189.004,142.746,-53.951,-178.375,6.257,148.651
C01429=1188.998,142.996,-53.972,-178.373,6.258,148.651
C01430=1188.994,143.245,-53.992,-178.370,6.260,148.650
C01431=1188.989,143.495,-54.013,-178.367,6.262,148.650
C01432=1188.985,143.744,-54.034,-178.365,6.263,148.650
C01433=1188.980,143.993,-54.055,-178.362,6.265,148.649
C01434=1188.975,144.242,-54.075,-178.360,6.266,148.649
C01435=1188.970,144.490,-54.097,-178.357,6.267,148.648
C01436=1188.966,144.739,-54.117,-178.354,6.269,148.648
C01437=1188.961,144.989,-54.138,-178.351,6.271,148.647
C01438=1188.956,145.238,-54.158,-178.349,6.272,148.647
C01439=1188.951,145.487,-54.179,-178.346,6.273,148.646
C01440=1188.947,145.736,-54.200,-178.343,6.275,148.646
C01441=1188.942,145.985,-54.221,-178.341,6.277,148.646
C01442=1188.937,146.234,-54.241,-178.339,6.278,148.645
C01443=1188.932,146.483,-54.263,-178.336,6.280,148.645
C01444=1188.929,146.732,-54.284,-178.333,6.281,148.644
C01445=1188.923,146.982,-54.305,-178.330,6.283,148.644
C01446=1188.919,147.231,-54.325,-178.327,6.285,148.644
C01447=1188.914,147.480,-54.346,-178.325,6.286,148.643
C01448=1188.910,147.728,-54.367,-178.323,6.287,148.643
C01449=1188.904,147.977,-54.388,-178.320,6.289,148.642
C01450=1188.899,148.227,-54.409,-178.317,6.290,148.642
C01451=1188.895,148.476,-54.429,-178.314,6.292,148.641
C01452=1188.890,148.726,-54.451,-178.312,6.293,148.641
C01453=1188.886,148.974,-54.472,-178.309,6.295,148.641
C01454=1188.881,149.223,-54.493,-178.307,6.297,148.640
C01455=1188.876,149.472,-54.514,-178.304,6.299,148.640
C01456=1188.872,149.721,-54.535,-178.301,6.300,148.639
C01457=1188.866,149.970,-54.556,-178.299,6.301,148.639
C01458=1188.861,150.219,-54.577,-178.296,6.303,148.638
C01459=1188.858,150.468,-54.598,-178.293,6.304,148.638
C01460=1188.853,150.718,-54.619,-178.291,6.306,148.638
C01461=1188.847,150.967,-54.640,-178.288,6.308,148.637
C01462=1188.843,151.215,-54.661,-178.285,6.309,148.637
C01463=1188.838,151.464,-54.682,-178.283,6.310,148.636
C01464=1188.834,151.714,-54.703,-178.280,6.312,148.636
C01465=1188.829,151.963,-54.724,-178.277,6.314,148.636
C01466=1188.824,152.212,-54.745,-178.275,6.316,148.635
C01467=1188.819,152.461,-54.767,-178.272,6.317,148.635
C01468=1188.814,152.710,-54.788,-178.270,6.318,148.634
C01469=1188.810,152.960,-54.809,-178.267,6.320,148.634
C01470=1188.805,153.208,-54.831,-178.264,6.322,148.633
C01471=1188.800,153.457,-54.851,-178.261,6.323,148.633
C01472=1188.795,153.706,-54.873,-178.259,6.325,148.633
C01473=1188.791,153.955,-54.894,-178.256,6.327,148.632
C01474=1188.787,154.204,-54.916,-178.254,6.328,148.632
C01475=1188.782,154.454,-54.937,-178.251,6.330,148.632
C01476=1188.777,154.702,-54.958,-178.248,6.331,148.631
C01477=1188.772,154.951,-54.979,-178.245,6.333,148.631
C01478=1188.768,155.201,-55.001,-178.243,6.335,148.630
C01479=1188.763,155.450,-55.022,-178.240,6.336,148.630
C01480=1188.758,155.698,-55.043,-178.238,6.337,148.629
C01481=1188.753,155.947,-55.065,-178.235,6.339,148.629
C01482=1188.749,156.197,-55.086,-178.232,6.341,148.629
C01483=1188.744,156.445,-55.107,-178.230,6.343,148.628
C01484=1188.739,156.695,-55.128,-178.227,6.344,148.628
C01485=1188.735,156.944,-55.150,-178.224,6.346,148.627
C01486=1188.730,157.193,-55.171,-178.221,6.348,148.627
C01487=1188.725,157.442,-55.193,-178.219,6.349,148.627
C01488=1188.720,157.690,-55.215,-178.216,6.350,148.626
C01489=1188.716,157.940,-55.236,-178.214,6.352,148.626
C01490=1188.711,158.189,-55.257,-178.211,6.354,148.625
C01491=1188.706,158.458,-55.281,-178.208,6.356,148.625
C01492=1188.701,158.727,-55.304,-178.205,6.357,148.624
C01493=1188.696,158.996,-55.327,-178.203,6.359,148.624
C01494=1188.691,159.265,-55.350,-178.200,6.361,148.624
C01495=1188.686,159.514,-55.372,-178.197,6.362,148.623
C01496=1188.681,159.762,-55.394,-178.194,6.364,148.623
C01497=1188.677,160.012,-55.415,-178.191,6.366,148.622
C01498=1188.672,160.261,-55.437,-178.189,6.367,148.622
C01499=1188.668,160.510,-55.459,-178.186,6.369,148.622
C01500=1188.663,160.759,-55.480,-178.183,6.371,148.621
C01501=1188.658,161.008,-55.501,-178.181,6.372,148.621
C01502=1188.653,161.257,-55.523,-178.178,6.374,148.621
C01503=1188.648,161.506,-55.545,-178.176,6.375,148.620
C01504=1188.644,161.755,-55.567,-178.173,6.377,148.620
C01505=1188.639,162.004,-55.589,-178.170,6.379,148.619
C01506=1188.634,162.253,-55.610,-178.168,6.381,148.619
C01507=1188.630,162.503,-55.632,-178.165,6.383,148.619
C01508=1188.625,162.751,-55.653,-178.162,6.384,148.618
C01509=1188.620,163.000,-55.675,-178.159,6.386,148.618
C01510=1188.616,163.249,-55.697,-178.157,6.387,148.617
C01511=1188.611,163.498,-55.719,-178.154,6.389,148.617
C01512=1188.607,163.747,-55.741,-178.152,6.390,148.617
C01513=1188.602,163.996,-55.763,-178.149,6.392,148.616
C01514=1188.597,164.245,-55.784,-178.146,6.394,148.616
C01515=1188.593,164.494,-55.806,-178.144,6.396,148.615
C01516=1188.588,164.743,-55.827,-178.141,6.397,148.615
C01517=1188.583,164.992,-55.849,-178.138,6.399,148.615
C01518=1188.578,165.241,-55.871,-178.136,6.401,148.614
C01519=1188.574,165.490,-55.893,-178.133,6.403,148.614
C01520=1188.569,165.739,-55.915,-178.130,6.405,148.614
C01521=1188.564,165.989,-55.937,-178.128,6.406,148.613
C01522=1188.559,166.237,-55.959,-178.126,6.407,148.613
C01523=1188.555,166.487,-55.981,-178.123,6.409,148.613
C01524=1188.550,166.735,-56.003,-178.120,6.411,148.612
C01525=1188.545,166.984,-56.024,-178.117,6.412,148.612
C01526=1188.541,167.233,-56.047,-178.114,6.414,148.611
C01527=1188.537,167.481,-56.069,-178.112,6.416,148.611
C01528=1188.532,167.731,-56.092,-178.109,6.418,148.610
C01529=1188.527,167.980,-56.113,-178.106,6.419,148.610
C01530=1188.522,168.229,-56.135,-178.104,6.421,148.610
C01531=1188.518,168.478,-56.157,-178.101,6.423,148.609
C01532=1188.513,168.727,-56.179,-178.098,6.425,148.609
C01533=1188.508,168.976,-56.201,-178.096,6.427,148.609
C01534=1188.503,169.225,-56.223,-178.094,6.428,148.608
C01535=1188.499,169.474,-56.245,-178.091,6.429,148.608
C01536=1188.495,169.723,-56.268,-178.088,6.431,148.607
C01537=1188.490,169.971,-56.289,-178.086,6.433,148.607
C01538=1188.485,170.221,-56.312,-178.083,6.435,148.607
C01539=1188.480,170.470,-56.334,-178.080,6.436,148.606
C01540=1188.476,170.719,-56.356,-178.078,6.438,148.606
C01541=1188.472,170.968,-56.379,-178.075,6.440,148.606
C01542=1188.466,171.217,-56.401,-178.072,6.442,148.605
C01543=1188.462,171.466,-56.423,-178.069,6.444,148.605
C01544=1188.457,171.715,-56.445,-178.067,6.445,148.605
C01545=1188.453,171.963,-56.467,-178.064,6.447,148.604
C01546=1188.447,172.212,-56.490,-178.061,6.449,148.604
C01547=1188.443,172.462,-56.512,-178.059,6.451,148.603
C01548=1188.439,172.711,-56.534,-178.056,6.453,148.603
C01549=1188.433,172.959,-56.557,-178.053,6.454,148.603
C01550=1188.429,173.209,-56.579,-178.051,6.456,148.602
C01551=1188.424,173.457,-56.600,-178.048,6.458,148.602
C01552=1188.420,173.706,-56.624,-178.045,6.460,148.602
C01553=1188.415,173.956,-56.646,-178.043,6.461,148.601
C01554=1188.411,174.204,-56.668,-178.040,6.463,148.601
C01555=1188.406,174.453,-56.691,-178.037,6.465,148.601
C01556=1188.401,174.702,-56.713,-178.035,6.466,148.600
C01557=1188.397,174.951,-56.735,-178.033,6.468,148.600
C01558=1188.392,175.200,-56.758,-178.030,6.470,148.599
C01559=1188.387,175.449,-56.780,-178.027,6.471,148.599
C01560=1188.382,175.698,-56.803,-178.025,6.473,148.599
C01561=1188.378,175.947,-56.825,-178.022,6.475,148.598
C01562=1188.374,176.195,-56.847,-178.019,6.477,148.598
C01563=1188.369,176.445,-56.870,-178.017,6.478,148.598
C01564=1188.365,176.694,-56.893,-178.014,6.480,148.597
C01565=1188.359,176.943,-56.915,-178.011,6.482,148.597
C01566=1188.355,177.191,-56.938,-178.009,6.484,148.597
C01567=1188.350,177.441,-56.961,-178.006,6.486,148.596
C01568=1188.345,177.689,-56.983,-178.003,6.487,148.596
C01569=1188.341,177.938,-57.005,-178.001,6.489,148.596
C01570=1188.337,178.187,-57.028,-177.998,6.491,148.595
C01571=1188.332,178.436,-57.050,-177.995,6.493,148.595
C01572=1188.327,178.685,-57.073,-177.993,6.495,148.594
C01573=1188.323,178.934,-57.095,-177.990,6.496,148.594
C01574=1188.317,179.183,-57.118,-177.987,6.498,148.594
C01575=1188.313,179.432,-57.140,-177.985,6.500,148.593
C01576=1188.308,179.681,-57.164,-177.982,6.502,148.593
C01577=1188.304,179.929,-57.186,-177.979,6.504,148.593
C01578=1188.299,180.179,-57.209,-177.977,6.505,148.592
C01579=1188.295,180.428,-57.232,-177.974,6.507,148.592
C01580=1188.290,180.677,-57.255,-177.972,6.509,148.592
C01581=1188.285,180.926,-57.277,-177.969,6.511,148.591
C01582=1188.281,181.174,-57.300,-177.966,6.513,148.591
C01583=1188.276,181.423,-57.323,-177.964,6.515,148.591
C01584=1188.272,181.673,-57.345,-177.961,6.516,148.590
C01585=1188.266,181.921,-57.368,-177.958,6.518,148.590
C01586=1188.262,182.170,-57.391,-177.955,6.521,148.590
C01587=1188.257,182.419,-57.414,-177.952,6.523,148.589
C01588=1188.253,182.668,-57.437,-177.950,6.524,148.589
C01589=1188.249,182.917,-57.460,-177.947,6.526,148.589
C01590=1188.243,183.165,-57.483,-177.944,6.528,148.588
C01591=1188.239,183.415,-57.505,-177.942,6.530,148.588
C01592=1188.234,183.664,-57.528,-177.939,6.532,148.588
C01593=1188.230,183.913,-57.552,-177.936,6.533,148.587
C01594=1188.225,184.161,-57.574,-177.934,6.535,148.587
C01595=1188.220,184.431,-57.599,-177.931,6.537,148.586
C01596=1188.215,184.700,-57.624,-177.928,6.539,148.586
C01597=1188.210,184.970,-57.649,-177.925,6.541,148.586
C01598=1188.205,185.240,-57.674,-177.922,6.543,148.585
C01599=1188.201,185.488,-57.696,-177.920,6.545,148.585
C01600=1188.196,185.737,-57.720,-177.917,6.547,148.585
C01601=1188.191,185.986,-57.743,-177.914,6.548,148.584
C01602=1188.187,186.235,-57.767,-177.912,6.550,148.584
C01603=1188.183,186.484,-57.789,-177.909,6.552,148.584
C01604=1188.177,186.733,-57.812,-177.907,6.554,148.583
C01605=1188.172,186.982,-57.835,-177.904,6.556,148.583
C01606=1188.168,187.231,-57.858,-177.902,6.558,148.583
C01607=1188.164,187.480,-57.881,-177.899,6.560,148.582
C01608=1188.159,187.729,-57.904,-177.896,6.562,148.582
C01609=1188.154,187.978,-57.928,-177.893,6.564,148.582
C01610=1188.150,188.227,-57.951,-177.890,6.566,148.581
C01611=1188.146,188.476,-57.974,-177.888,6.568,148.581
C01612=1188.140,188.724,-57.997,-177.885,6.569,148.581
C01613=1188.136,188.973,-58.020,-177.882,6.571,148.580
C01614=1188.131,189.222,-58.044,-177.880,6.573,148.580
C01615=1188.126,189.471,-58.067,-177.878,6.575,148.580
C01616=1188.122,189.720,-58.090,-177.875,6.577,148.579
C01617=1188.118,189.969,-58.113,-177.872,6.579,148.579
C01618=1188.113,190.218,-58.136,-177.870,6.580,148.579
C01619=1188.108,190.466,-58.161,-177.867,6.582,148.578
C01620=1188.104,190.715,-58.184,-177.864,6.584,148.578
C01621=1188.099,190.964,-58.207,-177.862,6.586,148.578
C01622=1188.094,191.212,-58.230,-177.858,6.588,148.577
C01623=1188.090,191.461,-58.253,-177.856,6.591,148.577
C01624=1188.085,191.710,-58.276,-177.853,6.592,148.577
C01625=1188.080,191.959,-58.300,-177.851,6.594,148.577
C01626=1188.076,192.209,-58.323,-177.848,6.596,148.576
C01627=1188.071,192.457,-58.347,-177.845,6.598,148.576
C01628=1188.067,192.706,-58.371,-177.843,6.600,148.576
C01629=1188.062,192.955,-58.394,-177.840,6.601,148.575
C01630=1188.057,193.204,-58.417,-177.838,6.604,148.575
C01631=1188.052,193.453,-58.441,-177.835,6.605,148.575
C01632=1188.049,193.701,-58.464,-177.832,6.608,148.574
C01633=1188.044,193.950,-58.487,-177.829,6.610,148.574
C01634=1188.039,194.199,-58.511,-177.827,6.612,148.574
C01635=1188.035,194.448,-58.534,-177.824,6.613,148.573
C01636=1188.030,194.697,-58.558,-177.821,6.615,148.573
C01637=1188.026,194.946,-58.582,-177.819,6.617,148.573
C01638=1188.021,195.195,-58.605,-177.817,6.619,148.572
C01639=1188.017,195.443,-58.629,-177.814,6.621,148.572
C01640=1188.012,195.692,-58.652,-177.811,6.623,148.572
C01641=1188.007,195.941,-58.676,-177.808,6.625,148.571
C01642=1188.003,196.190,-58.700,-177.805,6.627,148.571
C01643=1187.998,196.439,-58.723,-177.803,6.629,148.571
C01644=1187.993,196.688,-58.747,-177.801,6.631,148.571
C01645=1187.989,196.936,-58.771,-177.798,6.633,148.570
C01646=1187.984,197.185,-58.794,-177.795,6.635,148.570
C01647=1187.980,197.434,-58.817,-177.793,6.636,148.570
C01648=1187.974,197.683,-58.842,-177.790,6.638,148.569
C01649=1187.970,197.932,-58.865,-177.787,6.641,148.569
C01650=1187.965,198.180,-58.889,-177.784,6.643,148.569
C01651=1187.961,198.429,-58.913,-177.782,6.645,148.568
C01652=1187.956,198.678,-58.937,-177.779,6.647,148.568
C01653=1187.952,198.928,-58.961,-177.776,6.648,148.568
C01654=1187.948,199.176,-58.985,-177.774,6.650,148.567
C01655=1187.943,199.425,-59.008,-177.772,6.652,148.567
C01656=1187.939,199.673,-59.032,-177.768,6.655,148.567
C01657=1187.934,199.922,-59.055,-177.766,6.657,148.567
C01658=1187.930,200.171,-59.080,-177.763,6.659,148.566
C01659=1187.924,200.420,-59.103,-177.760,6.660,148.566
C01660=1187.920,200.669,-59.128,-177.758,6.662,148.566
C01661=1187.915,200.918,-59.151,-177.756,6.664,148.565
C01662=1187.911,201.166,-59.175,-177.753,6.666,148.565
C01663=1187.907,201.416,-59.199,-177.750,6.669,148.565
C01664=1187.902,201.664,-59.223,-177.747,6.671,148.564
C01665=1187.897,201.913,-59.247,-177.744,6.672,148.564
C01666=1187.892,202.162,-59.271,-177.742,6.674,148.564
C01667=1187.888,202.410,-59.295,-177.740,6.676,148.564
C01668=1187.883,202.659,-59.319,-177.737,6.678,148.563
C01669=1187.879,202.908,-59.342,-177.734,6.681,148.563
C01670=1187.874,203.157,-59.367,-177.731,6.683,148.563
C01671=1187.870,203.406,-59.391,-177.729,6.685,148.563
C01672=1187.865,203.655,-59.415,-177.726,6.686,148.562
C01673=1187.861,203.903,-59.439,-177.723,6.688,148.562
C01674=1187.856,204.152,-59.464,-177.721,6.690,148.562
C01675=1187.852,204.402,-59.487,-177.718,6.693,148.561
C01676=1187.847,204.650,-59.511,-177.715,6.695,148.561
C01677=1187.843,204.898,-59.535,-177.713,6.697,148.561
C01678=1187.838,205.147,-59.560,-177.710,6.698,148.560
C01679=1187.833,205.396,-59.583,-177.707,6.700,148.560
C01680=1187.829,205.645,-59.608,-177.705,6.703,148.560
C01681=1187.824,205.894,-59.633,-177.702,6.705,148.560
C01682=1187.820,206.142,-59.657,-177.699,6.707,148.559
C01683=1187.815,206.391,-59.681,-177.697,6.709,148.559
C01684=1187.810,206.640,-59.705,-177.695,6.711,148.559
C01685=1187.806,206.889,-59.729,-177.691,6.713,148.558
C01686=1187.802,207.138,-59.753,-177.689,6.715,148.558
C01687=1187.796,207.386,-59.778,-177.686,6.717,148.558
C01688=1187.792,207.635,-59.802,-177.684,6.719,148.558
C01689=1187.788,207.884,-59.826,-177.681,6.721,148.557
C01690=1187.783,208.133,-59.851,-177.678,6.724,148.557
C01691=1187.778,208.382,-59.874,-177.675,6.725,148.557
C01692=1187.773,208.630,-59.899,-177.673,6.727,148.556
C01693=1187.770,208.879,-59.923,-177.670,6.729,148.556
C01694=1187.765,209.128,-59.948,-177.668,6.731,148.556
C01695=1187.760,209.377,-59.972,-177.665,6.734,148.556
C01696=1187.756,209.625,-59.996,-177.662,6.736,148.555
C01697=1187.751,209.874,-60.021,-177.660,6.738,148.555
C01698=1187.747,210.123,-60.045,-177.657,6.740,148.555
C01699=1187.742,210.393,-60.072,-177.654,6.742,148.554
C01700=1187.736,210.663,-60.099,-177.651,6.744,148.554
C01701=1187.732,210.934,-60.126,-177.648,6.747,148.554
C01702=1187.726,211.205,-60.152,-177.645,6.748,148.553
C01703=1187.722,211.453,-60.176,-177.643,6.751,148.553
C01704=1187.717,211.703,-60.201,-177.640,6.753,148.553
C01705=1187.713,211.950,-60.226,-177.637,6.755,148.553
C01706=1187.708,212.199,-60.250,-177.635,6.757,148.553
C01707=1187.704,212.448,-60.275,-177.632,6.759,148.552
C01708=1187.699,212.697,-60.300,-177.629,6.762,148.552
C01709=1187.695,212.945,-60.324,-177.627,6.763,148.552
C01710=1187.690,213.195,-60.349,-177.624,6.766,148.552
C01711=1187.686,213.443,-60.373,-177.622,6.767,148.551
C01712=1187.681,213.692,-60.397,-177.618,6.770,148.551
C01713=1187.677,213.941,-60.423,-177.616,6.772,148.551
C01714=1187.672,214.189,-60.447,-177.614,6.774,148.550
C01715=1187.668,214.438,-60.472,-177.611,6.776,148.550
C01716=1187.663,214.687,-60.496,-177.608,6.778,148.550
C01717=1187.658,214.936,-60.521,-177.606,6.781,148.550
C01718=1187.655,215.184,-60.546,-177.603,6.782,148.549
C01719=1187.650,215.433,-60.571,-177.600,6.784,148.549
C01720=1187.646,215.682,-60.595,-177.598,6.787,148.549
C01721=1187.641,215.931,-60.620,-177.595,6.789,148.549
C01722=1187.636,216.179,-60.645,-177.592,6.791,148.548
C01723=1187.632,216.428,-60.670,-177.590,6.793,148.548
C01724=1187.627,216.677,-60.694,-177.587,6.796,148.548
C01725=1187.622,216.926,-60.719,-177.584,6.797,148.547
C01726=1187.618,217.174,-60.744,-177.582,6.799,148.547
C01727=1187.613,217.423,-60.769,-177.579,6.801,148.547
C01728=1187.609,217.672,-60.794,-177.576,6.804,148.547
C01729=1187.604,217.920,-60.819,-177.573,6.806,148.546
C01730=1187.600,218.169,-60.844,-177.571,6.808,148.546
C01731=1187.595,218.418,-60.868,-177.568,6.811,148.546
C01732=1187.591,218.667,-60.894,-177.565,6.812,148.546
C01733=1187.586,218.915,-60.918,-177.563,6.814,148.546
C01734=1187.582,219.164,-60.944,-177.561,6.816,148.545
C01735=1187.577,219.413,-60.969,-177.557,6.819,148.545
C01736=1187.573,219.661,-60.994,-177.555,6.821,148.545
C01737=1187.568,219.910,-61.019,-177.553,6.823,148.544
C01738=1187.564,220.159,-61.044,-177.550,6.825,148.544
C01739=1187.559,220.408,-61.069,-177.547,6.828,148.544
C01740=1187.555,220.657,-61.093,-177.545,6.829,148.544
C01741=1187.550,220.905,-61.119,-177.542,6.831,148.543
C01742=1187.546,221.154,-61.144,-177.539,6.834,148.543
C01743=1187.541,221.402,-61.169,-177.536,6.836,148.543
C01744=1187.537,221.651,-61.194,-177.534,6.838,148.543
C01745=1187.532,221.900,-61.219,-177.532,6.840,148.543
C01746=1187.528,222.148,-61.245,-177.528,6.843,148.542
C01747=1187.523,222.397,-61.269,-177.526,6.845,148.542
C01748=1187.519,222.646,-61.295,-177.524,6.847,148.542
C01749=1187.514,222.895,-61.320,-177.520,6.849,148.541
C01750=1187.510,223.143,-61.345,-177.518,6.851,148.541
C01751=1187.505,223.392,-61.370,-177.516,6.853,148.541
C01752=1187.501,223.641,-61.395,-177.512,6.856,148.541
C01753=1187.496,223.889,-61.421,-177.510,6.858,148.541
C01754=1187.491,224.138,-61.446,-177.508,6.860,148.540
C01755=1187.487,224.387,-61.472,-177.505,6.862,148.540
C01756=1187.482,224.635,-61.497,-177.502,6.865,148.540
C01757=1187.478,224.885,-61.522,-177.500,6.866,148.540
C01758=1187.473,225.133,-61.547,-177.497,6.869,148.539
C01759=1187.469,225.381,-61.573,-177.494,6.871,148.539
C01760=1187.465,225.629,-61.598,-177.491,6.873,148.539
C01761=1187.460,225.879,-61.623,-177.489,6.875,148.539
C01762=1187.456,226.127,-61.649,-177.486,6.878,148.538
C01763=1187.451,226.376,-61.674,-177.484,6.880,148.538
C01764=1187.447,226.624,-61.700,-177.481,6.882,148.538
C01765=1187.442,226.874,-61.725,-177.478,6.884,148.538
C01766=1187.437,227.122,-61.750,-177.476,6.887,148.538
C01767=1187.433,227.371,-61.776,-177.473,6.888,148.537
C01768=1187.428,227.619,-61.801,-177.470,6.891,148.537
C01769=1187.424,227.868,-61.827,-177.468,6.893,148.537
C01770=1187.420,228.117,-61.852,-177.465,6.895,148.537
C01771=1187.415,228.365,-61.878,-177.462,6.898,148.536
C01772=1187.411,228.614,-61.903,-177.460,6.900,148.536
C01773=1187.406,228.863,-61.929,-177.458,6.902,148.536
C01774=1187.402,229.111,-61.955,-177.454,6.905,148.536
C01775=1187.397,229.360,-61.980,-177.452,6.907,148.536
C01776=1187.393,229.608,-62.006,-177.450,6.909,148.535
C01777=1187.388,229.857,-62.031,-177.446,6.911,148.535
C01778=1187.384,230.106,-62.056,-177.444,6.913,148.535
C01779=1187.380,230.355,-62.082,-177.442,6.915,148.535
C01780=1187.374,230.603,-62.108,-177.439,6.918,148.534
C01781=1187.370,230.852,-62.134,-177.436,6.920,148.534
C01782=1187.366,231.101,-62.160,-177.434,6.922,148.534
C01783=1187.361,231.349,-62.185,-177.431,6.925,148.534
C01784=1187.356,231.598,-62.211,-177.429,6.927,148.534
C01785=1187.352,231.846,-62.237,-177.426,6.929,148.533
C01786=1187.348,232.095,-62.262,-177.423,6.931,148.533
C01787=1187.343,232.343,-62.288,-177.421,6.934,148.533
C01788=1187.339,232.592,-62.313,-177.418,6.935,148.533
C01789=1187.334,232.841,-62.340,-177.415,6.938,148.533
C01790=1187.330,233.090,-62.366,-177.413,6.940,148.532
C01791=1187.325,233.338,-62.392,-177.410,6.943,148.532
C01792=1187.321,233.586,-62.417,-177.407,6.945,148.532
C01793=1187.317,233.835,-62.443,-177.405,6.947,148.532
C01794=1187.312,234.084,-62.469,-177.402,6.950,148.531
C01795=1187.307,234.332,-62.495,-177.400,6.952,148.531
C01796=1187.303,234.581,-62.521,-177.397,6.954,148.531
C01797=1187.299,234.830,-62.546,-177.394,6.957,148.531
C01798=1187.295,235.078,-62.573,-177.392,6.959,148.531
C01799=1187.289,235.327,-62.599,-177.389,6.962,148.531
C01800=1187.285,235.575,-62.625,-177.386,6.963,148.530
C01801=1187.281,235.824,-62.650,-177.384,6.965,148.530
C01802=1187.276,236.073,-62.676,-177.381,6.968,148.530
C01803=1187.271,236.344,-62.705,-177.378,6.970,148.529
C01804=1187.266,236.616,-62.733,-177.375,6.973,148.529
C01805=1187.262,236.887,-62.762,-177.372,6.976,148.529
C01806=1187.257,237.159,-62.790,-177.370,6.978,148.529
C01807=1187.252,237.408,-62.816,-177.367,6.980,148.529
C01808=1187.247,237.656,-62.842,-177.365,6.983,148.529
C01809=1187.243,237.904,-62.868,-177.362,6.985,148.528
C01810=1187.238,238.154,-62.894,-177.359,6.987,148.528
C01811=1187.234,238.402,-62.921,-177.357,6.989,148.528
C01812=1187.230,238.651,-62.947,-177.354,6.992,148.528
C01813=1187.225,238.900,-62.973,-177.351,6.994,148.528
C01814=1187.221,239.148,-62.999,-177.349,6.997,148.527
C01815=1187.216,239.396,-63.025,-177.346,6.999,148.527
C01816=1187.212,239.644,-63.052,-177.344,7.001,148.527
C01817=1187.208,239.893,-63.078,-177.341,7.004,148.527
C01818=1187.203,240.142,-63.103,-177.338,7.006,148.527
C01819=1187.199,240.391,-63.130,-177.335,7.008,148.526
C01820=1187.194,240.639,-63.156,-177.333,7.011,148.526
C01821=1187.190,240.888,-63.183,-177.330,7.013,148.526
C01822=1187.186,241.137,-63.209,-177.328,7.015,148.526
C01823=1187.181,241.384,-63.235,-177.325,7.017,148.526
C01824=1187.176,241.633,-63.261,-177.322,7.020,148.526
C01825=1187.172,241.881,-63.288,-177.320,7.022,148.525
C01826=1187.167,242.131,-63.314,-177.317,7.025,148.525
C01827=1187.163,242.379,-63.341,-177.315,7.027,148.525
C01828=1187.158,242.628,-63.367,-177.312,7.030,148.525
